LIN {X 0,Y 387.487,Z 857.847,A -85,B 0,C 180,E1 10707.766,E2 10707.766} C_VEL
LIN {X 0,Y 387.621,Z 857.87,A -85,B 0,C 180,E1 10712.229,E2 10712.229} C_VEL
LIN {X 0,Y 387.482,Z 853.741,A -85,B 0,C 180,E1 10716.707,E2 10716.707} C_VEL
LIN {X 0,Y 387.632,Z 843.932,A -85,B 0,C 180,E1 10721.771,E2 10721.771} C_VEL
LIN {X 0,Y 388.622,Z 828.082,A -85,B 0,C 180,E1 10726.928,E2 10726.928} C_VEL
LIN {X 0,Y 390.979,Z 806.956,A -85,B 0,C 180,E1 10731.776,E2 10731.776} C_VEL
LIN {X 0,Y 394.767,Z 780.131,A -85,B 0,C 180,E1 10736.283,E2 10736.283} C_VEL
LIN {X 0,Y 399.363,Z 749.623,A -85,B 0,C 180,E1 10740.039,E2 10740.039} C_VEL
LIN {X 0,Y 404.501,Z 714.96,A -85,B 0,C 180,E1 10743.113,E2 10743.113} C_VEL
LIN {X 0,Y 409.027,Z 678.744,A -85,B 0,C 180,E1 10745.277,E2 10745.277} C_VEL
LIN {X 0,Y 411.733,Z 641.8,A -85,B 0,C 180,E1 10746.674,E2 10746.674} C_VEL
LIN {X 0,Y 397.961,Z 607.635,A -85,B 0,C 180,E1 10748.876,E2 10748.876} C_VEL
LIN {X 0,Y 385.205,Z 581.988,A -85,B 0,C 180,E1 10750.882,E2 10750.882} C_VEL
LIN {X 0,Y 385.096,Z 580.66,A -85,B 0,C 180,E1 10750.941,E2 10750.941} C_VEL
LIN {X 0,Y 385.068,Z 580.66,A -85,B 0,C 180,E1 10758.225,E2 10758.225} C_VEL
LIN {X 0,Y 385.156,Z 580.66,A -85,B 0,C 180,E1 10764.006,E2 10764.006} C_VEL
LIN {X 0,Y 385.319,Z 580.66,A -85,B 0,C 180,E1 10771.967,E2 10771.967} C_VEL
LIN {X 0,Y 385.586,Z 580.66,A -85,B 0,C 180,E1 10779.375,E2 10779.375} C_VEL
LIN {X 0,Y 385.8,Z 580.66,A -85,B 0,C 180,E1 10786.424,E2 10786.424} C_VEL
LIN {X 0,Y 386.219,Z 580.66,A -85,B 0,C 180,E1 10793.265,E2 10793.265} C_VEL
LIN {X 0,Y 386.491,Z 580.66,A -85,B 0,C 180,E1 10799.996,E2 10799.996} C_VEL
LIN {X 0,Y 386.22,Z 580.66,A -85,B 0,C 180,E1 10806.726,E2 10806.726} C_VEL
LIN {X 0,Y 385.936,Z 580.66,A -85,B 0,C 180,E1 10813.562,E2 10813.562} C_VEL
LIN {X 0,Y 385.606,Z 580.66,A -85,B 0,C 180,E1 10820.615,E2 10820.615} C_VEL
LIN {X 0,Y 385.322,Z 580.66,A -85,B 0,C 180,E1 10828.023,E2 10828.023} C_VEL
LIN {X 0,Y 385.109,Z 580.66,A -85,B 0,C 180,E1 10835.989,E2 10835.989} C_VEL
LIN {X 0,Y 385.017,Z 580.66,A -85,B 0,C 180,E1 10841.876,E2 10841.876} C_VEL
LIN {X 0,Y 385.076,Z 580.66,A -85,B 0,C 180,E1 10848.233,E2 10848.233} C_VEL
LIN {X 0,Y 385.211,Z 580.66,A -85,B 0,C 180,E1 10855.382,E2 10855.382} C_VEL
LIN {X 0,Y 398.177,Z 612.723,A -85,B 0,C 180,E1 10858.695,E2 10858.695} C_VEL
LIN {X 0,Y 406.244,Z 641.573,A -85,B 0,C 180,E1 10862.092,E2 10862.092} C_VEL
LIN {X 0,Y 406.168,Z 649.478,A -85,B 0,C 180,E1 10862.96,E2 10862.96} C_VEL
LIN {X 0,Y 401.431,Z 676.101,A -85,B 0,C 180,E1 10866.169,E2 10866.169} C_VEL
LIN {X 0,Y 396.838,Z 698.417,A -85,B 0,C 180,E1 10869.99,E2 10869.99} C_VEL
LIN {X 0,Y 392.904,Z 716.536,A -85,B 0,C 180,E1 10874.407,E2 10874.407} C_VEL
LIN {X 0,Y 390.375,Z 728.782,A -85,B 0,C 180,E1 10878.859,E2 10878.859} C_VEL
LIN {X 0,Y 389.058,Z 736.422,A -85,B 0,C 180,E1 10883.32,E2 10883.32} C_VEL
LIN {X 0,Y 388.574,Z 740.057,A -85,B 0,C 180,E1 10887.776,E2 10887.776} C_VEL
LIN {X 0,Y 388.582,Z 740.014,A -85,B 0,C 180,E1 10892.227,E2 10892.227} C_VEL
LIN {X 0,Y 389.15,Z 736.281,A -85,B 0,C 180,E1 10896.682,E2 10896.682} C_VEL
LIN {X 0,Y 390.68,Z 727.322,A -85,B 0,C 180,E1 10901.701,E2 10901.701} C_VEL
LIN {X 0,Y 393.773,Z 712.297,A -85,B 0,C 180,E1 10906.689,E2 10906.689} C_VEL
LIN {X 0,Y 398.048,Z 692.52,A -85,B 0,C 180,E1 10911.054,E2 10911.054} C_VEL
LIN {X 0,Y 402.806,Z 668.479,A -85,B 0,C 180,E1 10914.779,E2 10914.779} C_VEL
LIN {X 0,Y 406.697,Z 643.345,A -85,B 0,C 180,E1 10917.577,E2 10917.577} C_VEL
LIN {X 0,Y 398.963,Z 615.178,A -85,B 0,C 180,E1 10920.925,E2 10920.925} C_VEL
LIN {X 0,Y 386.913,Z 585.522,A -85,B 0,C 180,E1 10924.088,E2 10924.088} C_VEL
LIN {X 0,Y 385.16,Z 580.66,A -85,B 0,C 180,E1 10924.654,E2 10924.654} C_VEL
LIN {X 0,Y 385.049,Z 580.66,A -85,B 0,C 180,E1 10931.776,E2 10931.776} C_VEL
LIN {X 0,Y 385.058,Z 580.66,A -85,B 0,C 180,E1 10938.235,E2 10938.235} C_VEL
LIN {X 0,Y 385.139,Z 580.66,A -85,B 0,C 180,E1 10944.014,E2 10944.014} C_VEL
LIN {X 0,Y 385.264,Z 580.66,A -85,B 0,C 180,E1 10951.972,E2 10951.972} C_VEL
LIN {X 0,Y 385.581,Z 580.66,A -85,B 0,C 180,E1 10959.383,E2 10959.383} C_VEL
LIN {X 0,Y 385.746,Z 580.66,A -85,B 0,C 180,E1 10966.431,E2 10966.431} C_VEL
LIN {X 0,Y 386.233,Z 580.66,A -85,B 0,C 180,E1 10973.274,E2 10973.274} C_VEL
LIN {X 0,Y 386.501,Z 580.66,A -85,B 0,C 180,E1 10980.004,E2 10980.004} C_VEL
LIN {X 0,Y 386.216,Z 580.66,A -85,B 0,C 180,E1 10986.735,E2 10986.735} C_VEL
LIN {X 0,Y 385.929,Z 580.66,A -85,B 0,C 180,E1 10993.571,E2 10993.571} C_VEL
LIN {X 0,Y 385.585,Z 580.66,A -85,B 0,C 180,E1 11000.626,E2 11000.626} C_VEL
LIN {X 0,Y 385.302,Z 580.66,A -85,B 0,C 180,E1 11008.034,E2 11008.034} C_VEL
LIN {X 0,Y 385.067,Z 580.66,A -85,B 0,C 180,E1 11014.62,E2 11014.62} C_VEL
LIN {X 0,Y 385.011,Z 580.66,A -85,B 0,C 180,E1 11021.782,E2 11021.782} C_VEL
LIN {X 0,Y 385.175,Z 580.66,A -85,B 0,C 180,E1 11029.063,E2 11029.063} C_VEL
LIN {X 0,Y 407.62,Z 629.809,A -85,B 0,C 180,E1 11032.612,E2 11032.612} C_VEL
LIN {X 0,Y 412.212,Z 644.181,A -85,B 0,C 180,E1 11033.455,E2 11033.455} C_VEL
LIN {X 0,Y 408.523,Z 682.741,A -85,B 0,C 180,E1 11034.911,E2 11034.911} C_VEL
LIN {X 0,Y 403.964,Z 718.267,A -85,B 0,C 180,E1 11037.144,E2 11037.144} C_VEL
LIN {X 0,Y 398.982,Z 752.199,A -85,B 0,C 180,E1 11040.237,E2 11040.237} C_VEL
LIN {X 0,Y 394.303,Z 783.048,A -85,B 0,C 180,E1 11044.15,E2 11044.15} C_VEL
LIN {X 0,Y 390.715,Z 809.2,A -85,B 0,C 180,E1 11048.674,E2 11048.674} C_VEL
LIN {X 0,Y 388.558,Z 830.209,A -85,B 0,C 180,E1 11053.646,E2 11053.646} C_VEL
LIN {X 0,Y 387.619,Z 845.23,A -85,B 0,C 180,E1 11058.774,E2 11058.774} C_VEL
LIN {X 0,Y 387.505,Z 852.985,A -85,B 0,C 180,E1 11062.805,E2 11062.805} C_VEL
LIN {X 0,Y 385.019,Z 855.196,A -85,B 0,C 180,E1 11064.686,E2 11064.686} C_VEL
LIN {X 0,Y 379.649,Z 856.7,A -85,B 0,C 180,E1 11067.891,E2 11067.891} C_VEL
LIN {X 0,Y 379.794,Z 856.679,A -85,B 0,C 180,E1 11072.275,E2 11072.275} C_VEL
LIN {X 0,Y 379.657,Z 852.534,A -85,B 0,C 180,E1 11076.846,E2 11076.846} C_VEL
LIN {X 0,Y 379.775,Z 842.813,A -85,B 0,C 180,E1 11081.967,E2 11081.967} C_VEL
LIN {X 0,Y 380.838,Z 827.231,A -85,B 0,C 180,E1 11087.164,E2 11087.164} C_VEL
LIN {X 0,Y 383.309,Z 806.131,A -85,B 0,C 180,E1 11092.126,E2 11092.126} C_VEL
LIN {X 0,Y 387.248,Z 779.805,A -85,B 0,C 180,E1 11096.668,E2 11096.668} C_VEL
LIN {X 0,Y 392.071,Z 749.47,A -85,B 0,C 180,E1 11100.497,E2 11100.497} C_VEL
LIN {X 0,Y 397.304,Z 715.923,A -85,B 0,C 180,E1 11103.556,E2 11103.556} C_VEL
LIN {X 0,Y 402.117,Z 679.727,A -85,B 0,C 180,E1 11105.805,E2 11105.805} C_VEL
LIN {X 0,Y 405.031,Z 644.006,A -85,B 0,C 180,E1 11107.216,E2 11107.216} C_VEL
LIN {X 0,Y 392.035,Z 611.501,A -85,B 0,C 180,E1 11109.406,E2 11109.406} C_VEL
LIN {X 0,Y 377.128,Z 580.66,A -85,B 0,C 180,E1 11111.91,E2 11111.91} C_VEL
LIN {X 0,Y 377.101,Z 580.66,A -85,B 0,C 180,E1 11119.484,E2 11119.484} C_VEL
LIN {X 0,Y 377.196,Z 580.66,A -85,B 0,C 180,E1 11125.937,E2 11125.937} C_VEL
LIN {X 0,Y 377.413,Z 580.66,A -85,B 0,C 180,E1 11133.906,E2 11133.906} C_VEL
LIN {X 0,Y 377.618,Z 580.66,A -85,B 0,C 180,E1 11138.919,E2 11138.919} C_VEL
LIN {X 0,Y 377.856,Z 580.66,A -85,B 0,C 180,E1 11146.133,E2 11146.133} C_VEL
LIN {X 0,Y 378.293,Z 580.66,A -85,B 0,C 180,E1 11153.123,E2 11153.123} C_VEL
LIN {X 0,Y 378.59,Z 580.66,A -85,B 0,C 180,E1 11159.996,E2 11159.996} C_VEL
LIN {X 0,Y 378.296,Z 580.66,A -85,B 0,C 180,E1 11166.868,E2 11166.868} C_VEL
LIN {X 0,Y 377.984,Z 580.66,A -85,B 0,C 180,E1 11173.853,E2 11173.853} C_VEL
LIN {X 0,Y 377.637,Z 580.66,A -85,B 0,C 180,E1 11181.071,E2 11181.071} C_VEL
LIN {X 0,Y 377.334,Z 580.66,A -85,B 0,C 180,E1 11188.671,E2 11188.671} C_VEL
LIN {X 0,Y 377.167,Z 580.66,A -85,B 0,C 180,E1 11194.056,E2 11194.056} C_VEL
LIN {X 0,Y 377.046,Z 580.66,A -85,B 0,C 180,E1 11200.506,E2 11200.506} C_VEL
LIN {X 0,Y 377.061,Z 580.66,A -85,B 0,C 180,E1 11207.135,E2 11207.135} C_VEL
LIN {X 0,Y 377.268,Z 581.284,A -85,B 0,C 180,E1 11214.461,E2 11214.461} C_VEL
LIN {X 0,Y 390.662,Z 613.094,A -85,B 0,C 180,E1 11217.911,E2 11217.911} C_VEL
LIN {X 0,Y 398.837,Z 642.106,A -85,B 0,C 180,E1 11221.418,E2 11221.418} C_VEL
LIN {X 0,Y 399.58,Z 649.041,A -85,B 0,C 180,E1 11222.269,E2 11222.269} C_VEL
LIN {X 0,Y 394.701,Z 675.471,A -85,B 0,C 180,E1 11225.436,E2 11225.436} C_VEL
LIN {X 0,Y 389.766,Z 698.393,A -85,B 0,C 180,E1 11229.334,E2 11229.334} C_VEL
LIN {X 0,Y 385.74,Z 716.002,A -85,B 0,C 180,E1 11233.577,E2 11233.577} C_VEL
LIN {X 0,Y 382.702,Z 729.982,A -85,B 0,C 180,E1 11238.632,E2 11238.632} C_VEL
LIN {X 0,Y 381.313,Z 737.611,A -85,B 0,C 180,E1 11243.184,E2 11243.184} C_VEL
LIN {X 0,Y 380.788,Z 741.241,A -85,B 0,C 180,E1 11247.731,E2 11247.731} C_VEL
LIN {X 0,Y 380.797,Z 741.198,A -85,B 0,C 180,E1 11252.273,E2 11252.273} C_VEL
LIN {X 0,Y 381.602,Z 736.01,A -85,B 0,C 180,E1 11257.918,E2 11257.918} C_VEL
LIN {X 0,Y 383.654,Z 725.73,A -85,B 0,C 180,E1 11263.072,E2 11263.072} C_VEL
LIN {X 0,Y 387.075,Z 710.25,A -85,B 0,C 180,E1 11267.876,E2 11267.876} C_VEL
LIN {X 0,Y 391.675,Z 689.835,A -85,B 0,C 180,E1 11272.192,E2 11272.192} C_VEL
LIN {X 0,Y 396.785,Z 664.357,A -85,B 0,C 180,E1 11275.936,E2 11275.936} C_VEL
LIN {X 0,Y 399.548,Z 645.168,A -85,B 0,C 180,E1 11278.079,E2 11278.079} C_VEL
LIN {X 0,Y 391.906,Z 617.092,A -85,B 0,C 180,E1 11281.529,E2 11281.529} C_VEL
LIN {X 0,Y 380.331,Z 588.674,A -85,B 0,C 180,E1 11284.708,E2 11284.708} C_VEL
LIN {X 0,Y 377.226,Z 580.66,A -85,B 0,C 180,E1 11285.614,E2 11285.614} C_VEL
LIN {X 0,Y 377.045,Z 580.66,A -85,B 0,C 180,E1 11292.872,E2 11292.872} C_VEL
LIN {X 0,Y 377.104,Z 580.66,A -85,B 0,C 180,E1 11300.2,E2 11300.2} C_VEL
LIN {X 0,Y 377.171,Z 580.66,A -85,B 0,C 180,E1 11307.157,E2 11307.157} C_VEL
LIN {X 0,Y 377.374,Z 580.66,A -85,B 0,C 180,E1 11313.913,E2 11313.913} C_VEL
LIN {X 0,Y 377.61,Z 580.66,A -85,B 0,C 180,E1 11318.928,E2 11318.928} C_VEL
LIN {X 0,Y 377.805,Z 580.66,A -85,B 0,C 180,E1 11326.14,E2 11326.14} C_VEL
LIN {X 0,Y 378.304,Z 580.66,A -85,B 0,C 180,E1 11333.155,E2 11333.155} C_VEL
LIN {X 0,Y 378.599,Z 580.66,A -85,B 0,C 180,E1 11340.004,E2 11340.004} C_VEL
LIN {X 0,Y 378.299,Z 580.66,A -85,B 0,C 180,E1 11346.877,E2 11346.877} C_VEL
LIN {X 0,Y 377.979,Z 580.66,A -85,B 0,C 180,E1 11353.862,E2 11353.862} C_VEL
LIN {X 0,Y 377.616,Z 580.66,A -85,B 0,C 180,E1 11361.081,E2 11361.081} C_VEL
LIN {X 0,Y 377.338,Z 580.66,A -85,B 0,C 180,E1 11368.68,E2 11368.68} C_VEL
LIN {X 0,Y 377.161,Z 580.66,A -85,B 0,C 180,E1 11374.067,E2 11374.067} C_VEL
LIN {X 0,Y 377.026,Z 580.66,A -85,B 0,C 180,E1 11380.497,E2 11380.497} C_VEL
LIN {X 0,Y 377.195,Z 580.872,A -85,B 0,C 180,E1 11388.16,E2 11388.16} C_VEL
LIN {X 0,Y 386.408,Z 599.748,A -85,B 0,C 180,E1 11389.706,E2 11389.706} C_VEL
LIN {X 0,Y 403.016,Z 637.674,A -85,B 0,C 180,E1 11392.386,E2 11392.386} C_VEL
LIN {X 0,Y 405.397,Z 647.401,A -85,B 0,C 180,E1 11392.942,E2 11392.942} C_VEL
LIN {X 0,Y 401.341,Z 685.437,A -85,B 0,C 180,E1 11394.49,E2 11394.49} C_VEL
LIN {X 0,Y 396.408,Z 721.378,A -85,B 0,C 180,E1 11396.873,E2 11396.873} C_VEL
LIN {X 0,Y 391.163,Z 755.108,A -85,B 0,C 180,E1 11400.13,E2 11400.13} C_VEL
LIN {X 0,Y 386.341,Z 785.338,A -85,B 0,C 180,E1 11404.188,E2 11404.188} C_VEL
LIN {X 0,Y 382.632,Z 811.449,A -85,B 0,C 180,E1 11408.978,E2 11408.978} C_VEL
LIN {X 0,Y 380.581,Z 830.851,A -85,B 0,C 180,E1 11413.885,E2 11413.885} C_VEL
LIN {X 0,Y 379.721,Z 845.274,A -85,B 0,C 180,E1 11419.118,E2 11419.118} C_VEL
LIN {X 0,Y 379.676,Z 852.977,A -85,B 0,C 180,E1 11423.511,E2 11423.511} C_VEL
LIN {X 0,Y 379.649,Z 856.7,A -85,B 0,C 180,E1 11427.891,E2 11427.891} C_VEL
LIN {X 0,Y 377.151,Z 856.83,A -85,B 0,C 180,E1 11429.837,E2 11429.837} C_VEL
LIN {X 0,Y 371.879,Z 854.962,A -85,B 0,C 180,E1 11433.101,E2 11433.101} C_VEL
LIN {X 0,Y 371.822,Z 849.562,A -85,B 0,C 180,E1 11438.164,E2 11438.164} C_VEL
LIN {X 0,Y 372.107,Z 838.206,A -85,B 0,C 180,E1 11443.558,E2 11443.558} C_VEL
LIN {X 0,Y 373.57,Z 821.118,A -85,B 0,C 180,E1 11448.85,E2 11448.85} C_VEL
LIN {X 0,Y 376.666,Z 798.023,A -85,B 0,C 180,E1 11453.927,E2 11453.927} C_VEL
LIN {X 0,Y 381.131,Z 770.539,A -85,B 0,C 180,E1 11458.363,E2 11458.363} C_VEL
LIN {X 0,Y 386.638,Z 738.34,A -85,B 0,C 180,E1 11462.121,E2 11462.121} C_VEL
LIN {X 0,Y 392.059,Z 704.385,A -85,B 0,C 180,E1 11464.934,E2 11464.934} C_VEL
LIN {X 0,Y 396.892,Z 667.975,A -85,B 0,C 180,E1 11466.93,E2 11466.93} C_VEL
LIN {X 0,Y 398.263,Z 645.749,A -85,B 0,C 180,E1 11467.803,E2 11467.803} C_VEL
LIN {X 0,Y 385.396,Z 613.636,A -85,B 0,C 180,E1 11470.079,E2 11470.079} C_VEL
LIN {X 0,Y 369.227,Z 581.844,A -85,B 0,C 180,E1 11472.825,E2 11472.825} C_VEL
LIN {X 0,Y 369.134,Z 580.66,A -85,B 0,C 180,E1 11472.996,E2 11472.996} C_VEL
LIN {X 0,Y 369.156,Z 580.66,A -85,B 0,C 180,E1 11479.152,E2 11479.152} C_VEL
LIN {X 0,Y 369.201,Z 580.66,A -85,B 0,C 180,E1 11485.094,E2 11485.094} C_VEL
LIN {X 0,Y 369.331,Z 580.66,A -85,B 0,C 180,E1 11490.638,E2 11490.638} C_VEL
LIN {X 0,Y 369.537,Z 580.66,A -85,B 0,C 180,E1 11495.896,E2 11495.896} C_VEL
LIN {X 0,Y 369.846,Z 580.66,A -85,B 0,C 180,E1 11503.402,E2 11503.402} C_VEL
LIN {X 0,Y 370.128,Z 580.66,A -85,B 0,C 180,E1 11510.611,E2 11510.611} C_VEL
LIN {X 0,Y 370.709,Z 580.66,A -85,B 0,C 180,E1 11517.663,E2 11517.663} C_VEL
LIN {X 0,Y 370.608,Z 580.66,A -85,B 0,C 180,E1 11524.666,E2 11524.666} C_VEL
LIN {X 0,Y 370.124,Z 580.66,A -85,B 0,C 180,E1 11531.932,E2 11531.932} C_VEL
LIN {X 0,Y 369.775,Z 580.66,A -85,B 0,C 180,E1 11539.048,E2 11539.048} C_VEL
LIN {X 0,Y 369.457,Z 580.66,A -85,B 0,C 180,E1 11546.69,E2 11546.69} C_VEL
LIN {X 0,Y 369.278,Z 580.66,A -85,B 0,C 180,E1 11552.08,E2 11552.08} C_VEL
LIN {X 0,Y 369.09,Z 580.66,A -85,B 0,C 180,E1 11559.038,E2 11559.038} C_VEL
LIN {X 0,Y 369.142,Z 580.66,A -85,B 0,C 180,E1 11565.984,E2 11565.984} C_VEL
LIN {X 0,Y 369.295,Z 580.686,A -85,B 0,C 180,E1 11573.414,E2 11573.414} C_VEL
LIN {X 0,Y 382.702,Z 612.445,A -85,B 0,C 180,E1 11576.965,E2 11576.965} C_VEL
LIN {X 0,Y 390.981,Z 640.632,A -85,B 0,C 180,E1 11580.443,E2 11580.443} C_VEL
LIN {X 0,Y 392.512,Z 651.519,A -85,B 0,C 180,E1 11581.853,E2 11581.853} C_VEL
LIN {X 0,Y 387.224,Z 678.672,A -85,B 0,C 180,E1 11585.237,E2 11585.237} C_VEL
LIN {X 0,Y 382.184,Z 700.911,A -85,B 0,C 180,E1 11589.188,E2 11589.188} C_VEL
LIN {X 0,Y 377.843,Z 718.965,A -85,B 0,C 180,E1 11593.769,E2 11593.769} C_VEL
LIN {X 0,Y 374.79,Z 732.393,A -85,B 0,C 180,E1 11598.977,E2 11598.977} C_VEL
LIN {X 0,Y 373.319,Z 740.078,A -85,B 0,C 180,E1 11604.202,E2 11604.202} C_VEL
LIN {X 0,Y 372.998,Z 742.425,A -85,B 0,C 180,E1 11607.683,E2 11607.683} C_VEL
LIN {X 0,Y 373.007,Z 742.383,A -85,B 0,C 180,E1 11612.32,E2 11612.32} C_VEL
LIN {X 0,Y 373.813,Z 737.617,A -85,B 0,C 180,E1 11617.804,E2 11617.804} C_VEL
LIN {X 0,Y 376.06,Z 726.932,A -85,B 0,C 180,E1 11623.341,E2 11623.341} C_VEL
LIN {X 0,Y 379.463,Z 712.313,A -85,B 0,C 180,E1 11628.022,E2 11628.022} C_VEL
LIN {X 0,Y 384.164,Z 692.319,A -85,B 0,C 180,E1 11632.405,E2 11632.405} C_VEL
LIN {X 0,Y 389.405,Z 667.874,A -85,B 0,C 180,E1 11636.155,E2 11636.155} C_VEL
LIN {X 0,Y 392.524,Z 647.521,A -85,B 0,C 180,E1 11638.527,E2 11638.527} C_VEL
LIN {X 0,Y 384.969,Z 619.184,A -85,B 0,C 180,E1 11642.131,E2 11642.131} C_VEL
LIN {X 0,Y 373.521,Z 590.683,A -85,B 0,C 180,E1 11645.441,E2 11645.441} C_VEL
LIN {X 0,Y 369.288,Z 580.66,A -85,B 0,C 180,E1 11646.597,E2 11646.597} C_VEL
LIN {X 0,Y 369.139,Z 580.66,A -85,B 0,C 180,E1 11654.022,E2 11654.022} C_VEL
LIN {X 0,Y 369.13,Z 580.66,A -85,B 0,C 180,E1 11660.96,E2 11660.96} C_VEL
LIN {X 0,Y 369.253,Z 580.66,A -85,B 0,C 180,E1 11667.918,E2 11667.918} C_VEL
LIN {X 0,Y 369.513,Z 580.66,A -85,B 0,C 180,E1 11675.904,E2 11675.904} C_VEL
LIN {X 0,Y 369.746,Z 580.66,A -85,B 0,C 180,E1 11680.95,E2 11680.95} C_VEL
LIN {X 0,Y 369.994,Z 580.66,A -85,B 0,C 180,E1 11688.239,E2 11688.239} C_VEL
LIN {X 0,Y 370.488,Z 580.66,A -85,B 0,C 180,E1 11695.332,E2 11695.332} C_VEL
LIN {X 0,Y 370.722,Z 580.66,A -85,B 0,C 180,E1 11700.004,E2 11700.004} C_VEL
LIN {X 0,Y 370.369,Z 580.66,A -85,B 0,C 180,E1 11707.025,E2 11707.025} C_VEL
LIN {X 0,Y 370.037,Z 580.66,A -85,B 0,C 180,E1 11714.166,E2 11714.166} C_VEL
LIN {X 0,Y 369.677,Z 580.66,A -85,B 0,C 180,E1 11721.556,E2 11721.556} C_VEL
LIN {X 0,Y 369.456,Z 580.66,A -85,B 0,C 180,E1 11726.7,E2 11726.7} C_VEL
LIN {X 0,Y 369.268,Z 580.66,A -85,B 0,C 180,E1 11732.091,E2 11732.091} C_VEL
LIN {X 0,Y 369.058,Z 580.66,A -85,B 0,C 180,E1 11739.026,E2 11739.026} C_VEL
LIN {X 0,Y 369.152,Z 580.66,A -85,B 0,C 180,E1 11745.98,E2 11745.98} C_VEL
LIN {X 0,Y 369.209,Z 581.4,A -85,B 0,C 180,E1 11747.179,E2 11747.179} C_VEL
LIN {X 0,Y 391.31,Z 626.732,A -85,B 0,C 180,E1 11750.903,E2 11750.903} C_VEL
LIN {X 0,Y 398.754,Z 648.256,A -85,B 0,C 180,E1 11752.346,E2 11752.346} C_VEL
LIN {X 0,Y 394.452,Z 686.258,A -85,B 0,C 180,E1 11753.954,E2 11753.954} C_VEL
LIN {X 0,Y 389.256,Z 722.076,A -85,B 0,C 180,E1 11756.401,E2 11756.401} C_VEL
LIN {X 0,Y 383.757,Z 755.406,A -85,B 0,C 180,E1 11759.728,E2 11759.728} C_VEL
LIN {X 0,Y 378.743,Z 785.057,A -85,B 0,C 180,E1 11763.818,E2 11763.818} C_VEL
LIN {X 0,Y 374.823,Z 811.132,A -85,B 0,C 180,E1 11768.756,E2 11768.756} C_VEL
LIN {X 0,Y 372.615,Z 831.492,A -85,B 0,C 180,E1 11774.135,E2 11774.135} C_VEL
LIN {X 0,Y 371.851,Z 845.324,A -85,B 0,C 180,E1 11779.477,E2 11779.477} C_VEL
LIN {X 0,Y 371.849,Z 852.304,A -85,B 0,C 180,E1 11783.824,E2 11783.824} C_VEL
LIN {X 0,Y 371.828,Z 855.519,A -85,B 0,C 180,E1 11787.884,E2 11787.884} C_VEL
LIN {X 0,Y 371.967,Z 855.488,A -85,B 0,C 180,E1 11792.323,E2 11792.323} C_VEL
LIN {X 0,Y 371.879,Z 854.962,A -85,B 0,C 180,E1 11793.101,E2 11793.101} C_VEL
LIN {X 0,Y 369.293,Z 853.192,A -85,B 0,C 180,E1 11795.068,E2 11795.068} C_VEL
LIN {X 0,Y 364.056,Z 848.87,A -85,B 0,C 180,E1 11797.999,E2 11797.999} C_VEL
LIN {X 0,Y 363.982,Z 848.354,A -85,B 0,C 180,E1 11798.338,E2 11798.338} C_VEL
LIN {X 0,Y 364.281,Z 836.657,A -85,B 0,C 180,E1 11803.975,E2 11803.975} C_VEL
LIN {X 0,Y 366.051,Z 818.641,A -85,B 0,C 180,E1 11809.566,E2 11809.566} C_VEL
LIN {X 0,Y 369.486,Z 795.121,A -85,B 0,C 180,E1 11814.744,E2 11814.744} C_VEL
LIN {X 0,Y 374.437,Z 766.272,A -85,B 0,C 180,E1 11819.346,E2 11819.346} C_VEL
LIN {X 0,Y 380.177,Z 733.933,A -85,B 0,C 180,E1 11823.073,E2 11823.073} C_VEL
LIN {X 0,Y 386.003,Z 698.709,A -85,B 0,C 180,E1 11825.897,E2 11825.897} C_VEL
LIN {X 0,Y 390.728,Z 663.112,A -85,B 0,C 180,E1 11827.761,E2 11827.761} C_VEL
LIN {X 0,Y 391.645,Z 647.863,A -85,B 0,C 180,E1 11828.377,E2 11828.377} C_VEL
LIN {X 0,Y 378.919,Z 616.13,A -85,B 0,C 180,E1 11830.754,E2 11830.754} C_VEL
LIN {X 0,Y 361.299,Z 581.694,A -85,B 0,C 180,E1 11833.878,E2 11833.878} C_VEL
LIN {X 0,Y 361.227,Z 580.66,A -85,B 0,C 180,E1 11833.994,E2 11833.994} C_VEL
LIN {X 0,Y 361.234,Z 580.66,A -85,B 0,C 180,E1 11841.199,E2 11841.199} C_VEL
LIN {X 0,Y 361.277,Z 580.66,A -85,B 0,C 180,E1 11847.111,E2 11847.111} C_VEL
LIN {X 0,Y 361.455,Z 580.66,A -85,B 0,C 180,E1 11852.66,E2 11852.66} C_VEL
LIN {X 0,Y 361.69,Z 580.66,A -85,B 0,C 180,E1 11857.943,E2 11857.943} C_VEL
LIN {X 0,Y 361.979,Z 580.66,A -85,B 0,C 180,E1 11865.512,E2 11865.512} C_VEL
LIN {X 0,Y 362.435,Z 580.66,A -85,B 0,C 180,E1 11872.821,E2 11872.821} C_VEL
LIN {X 0,Y 362.812,Z 580.66,A -85,B 0,C 180,E1 11879.996,E2 11879.996} C_VEL
LIN {X 0,Y 362.445,Z 580.66,A -85,B 0,C 180,E1 11887.17,E2 11887.17} C_VEL
LIN {X 0,Y 362.1,Z 580.66,A -85,B 0,C 180,E1 11894.474,E2 11894.474} C_VEL
LIN {X 0,Y 361.707,Z 580.66,A -85,B 0,C 180,E1 11902.046,E2 11902.046} C_VEL
LIN {X 0,Y 361.385,Z 580.66,A -85,B 0,C 180,E1 11908.742,E2 11908.742} C_VEL
LIN {X 0,Y 361.178,Z 580.66,A -85,B 0,C 180,E1 11915.788,E2 11915.788} C_VEL
LIN {X 0,Y 361.179,Z 580.66,A -85,B 0,C 180,E1 11921.939,E2 11921.939} C_VEL
LIN {X 0,Y 361.251,Z 580.66,A -85,B 0,C 180,E1 11928.741,E2 11928.741} C_VEL
LIN {X 0,Y 361.288,Z 580.699,A -85,B 0,C 180,E1 11932.329,E2 11932.329} C_VEL
LIN {X 0,Y 375.138,Z 612.697,A -85,B 0,C 180,E1 11936.083,E2 11936.083} C_VEL
LIN {X 0,Y 383.173,Z 639.476,A -85,B 0,C 180,E1 11939.471,E2 11939.471} C_VEL
LIN {X 0,Y 385.708,Z 652.742,A -85,B 0,C 180,E1 11941.292,E2 11941.292} C_VEL
LIN {X 0,Y 380.178,Z 679.949,A -85,B 0,C 180,E1 11944.746,E2 11944.746} C_VEL
LIN {X 0,Y 374.903,Z 702.152,A -85,B 0,C 180,E1 11948.765,E2 11948.765} C_VEL
LIN {X 0,Y 370.327,Z 720.178,A -85,B 0,C 180,E1 11953.43,E2 11953.43} C_VEL
LIN {X 0,Y 367.119,Z 733.591,A -85,B 0,C 180,E1 11958.744,E2 11958.744} C_VEL
LIN {X 0,Y 365.55,Z 741.266,A -85,B 0,C 180,E1 11964.079,E2 11964.079} C_VEL
LIN {X 0,Y 365.212,Z 743.609,A -85,B 0,C 180,E1 11967.634,E2 11967.634} C_VEL
LIN {X 0,Y 365.222,Z 743.567,A -85,B 0,C 180,E1 11972.37,E2 11972.37} C_VEL
LIN {X 0,Y 365.884,Z 739.855,A -85,B 0,C 180,E1 11977.109,E2 11977.109} C_VEL
LIN {X 0,Y 367.748,Z 730.936,A -85,B 0,C 180,E1 11982.442,E2 11982.442} C_VEL
LIN {X 0,Y 371.34,Z 716.166,A -85,B 0,C 180,E1 11987.666,E2 11987.666} C_VEL
LIN {X 0,Y 376.133,Z 697.11,A -85,B 0,C 180,E1 11992.177,E2 11992.177} C_VEL
LIN {X 0,Y 381.475,Z 673.599,A -85,B 0,C 180,E1 11996.079,E2 11996.079} C_VEL
LIN {X 0,Y 385.666,Z 650.724,A -85,B 0,C 180,E1 11998.858,E2 11998.858} C_VEL
LIN {X 0,Y 378.791,Z 623.486,A -85,B 0,C 180,E1 12002.486,E2 12002.486} C_VEL
LIN {X 0,Y 367.612,Z 594.962,A -85,B 0,C 180,E1 12005.96,E2 12005.96} C_VEL
LIN {X 0,Y 361.269,Z 580.66,A -85,B 0,C 180,E1 12007.578,E2 12007.578} C_VEL
LIN {X 0,Y 361.217,Z 580.66,A -85,B 0,C 180,E1 12015.249,E2 12015.249} C_VEL
LIN {X 0,Y 361.206,Z 580.66,A -85,B 0,C 180,E1 12022.537,E2 12022.537} C_VEL
LIN {X 0,Y 361.358,Z 580.66,A -85,B 0,C 180,E1 12029.935,E2 12029.935} C_VEL
LIN {X 0,Y 361.679,Z 580.66,A -85,B 0,C 180,E1 12037.952,E2 12037.952} C_VEL
LIN {X 0,Y 361.918,Z 580.66,A -85,B 0,C 180,E1 12045.519,E2 12045.519} C_VEL
LIN {X 0,Y 362.43,Z 580.66,A -85,B 0,C 180,E1 12053.135,E2 12053.135} C_VEL
LIN {X 0,Y 362.819,Z 580.66,A -85,B 0,C 180,E1 12060.004,E2 12060.004} C_VEL
LIN {X 0,Y 362.455,Z 580.66,A -85,B 0,C 180,E1 12067.179,E2 12067.179} C_VEL
LIN {X 0,Y 362.082,Z 580.66,A -85,B 0,C 180,E1 12074.484,E2 12074.484} C_VEL
LIN {X 0,Y 361.69,Z 580.66,A -85,B 0,C 180,E1 12082.057,E2 12082.057} C_VEL
LIN {X 0,Y 361.385,Z 580.66,A -85,B 0,C 180,E1 12090.073,E2 12090.073} C_VEL
LIN {X 0,Y 361.146,Z 580.66,A -85,B 0,C 180,E1 12097.45,E2 12097.45} C_VEL
LIN {X 0,Y 361.193,Z 580.66,A -85,B 0,C 180,E1 12104.747,E2 12104.747} C_VEL
LIN {X 0,Y 361.282,Z 581.215,A -85,B 0,C 180,E1 12106.126,E2 12106.126} C_VEL
LIN {X 0,Y 383.637,Z 626.463,A -85,B 0,C 180,E1 12110.068,E2 12110.068} C_VEL
LIN {X 0,Y 391.968,Z 649.234,A -85,B 0,C 180,E1 12111.726,E2 12111.726} C_VEL
LIN {X 0,Y 387.707,Z 686.192,A -85,B 0,C 180,E1 12113.347,E2 12113.347} C_VEL
LIN {X 0,Y 382.165,Z 722.435,A -85,B 0,C 180,E1 12115.886,E2 12115.886} C_VEL
LIN {X 0,Y 376.285,Z 756.1,A -85,B 0,C 180,E1 12119.356,E2 12119.356} C_VEL
LIN {X 0,Y 371.185,Z 784.787,A -85,B 0,C 180,E1 12123.436,E2 12123.436} C_VEL
LIN {X 0,Y 367.2,Z 809.818,A -85,B 0,C 180,E1 12128.293,E2 12128.293} C_VEL
LIN {X 0,Y 364.984,Z 828.294,A -85,B 0,C 180,E1 12133.176,E2 12133.176} C_VEL
LIN {X 0,Y 364.039,Z 842.803,A -85,B 0,C 180,E1 12138.643,E2 12138.643} C_VEL
LIN {X 0,Y 364.02,Z 850.112,A -85,B 0,C 180,E1 12142.855,E2 12142.855} C_VEL
LIN {X 0,Y 364.024,Z 854.276,A -85,B 0,C 180,E1 12147.622,E2 12147.622} C_VEL
LIN {X 0,Y 364.14,Z 854.297,A -85,B 0,C 180,E1 12152.373,E2 12152.373} C_VEL
LIN {X 0,Y 363.996,Z 850.12,A -85,B 0,C 180,E1 12157.142,E2 12157.142} C_VEL
LIN {X 0,Y 363.982,Z 848.354,A -85,B 0,C 180,E1 12158.338,E2 12158.338} C_VEL
LIN {X 0,Y 361.535,Z 844.791,A -85,B 0,C 180,E1 12160.295,E2 12160.295} C_VEL
LIN {X 0,Y 356.399,Z 838.109,A -85,B 0,C 180,E1 12163.178,E2 12163.178} C_VEL
LIN {X 0,Y 356.353,Z 837.297,A -85,B 0,C 180,E1 12163.509,E2 12163.509} C_VEL
LIN {X 0,Y 357.9,Z 820.394,A -85,B 0,C 180,E1 12169.186,E2 12169.186} C_VEL
LIN {X 0,Y 361.501,Z 796.939,A -85,B 0,C 180,E1 12174.668,E2 12174.668} C_VEL
LIN {X 0,Y 366.338,Z 769.814,A -85,B 0,C 180,E1 12179.281,E2 12179.281} C_VEL
LIN {X 0,Y 372.334,Z 738.262,A -85,B 0,C 180,E1 12183.166,E2 12183.166} C_VEL
LIN {X 0,Y 378.164,Z 705.17,A -85,B 0,C 180,E1 12186.051,E2 12186.051} C_VEL
LIN {X 0,Y 383.426,Z 669.623,A -85,B 0,C 180,E1 12188.129,E2 12188.129} C_VEL
LIN {X 0,Y 384.867,Z 649.638,A -85,B 0,C 180,E1 12188.992,E2 12188.992} C_VEL
LIN {X 0,Y 371.618,Z 616.677,A -85,B 0,C 180,E1 12191.611,E2 12191.611} C_VEL
LIN {X 0,Y 353.37,Z 581.449,A -85,B 0,C 180,E1 12195,E2 12195} C_VEL
LIN {X 0,Y 353.28,Z 580.66,A -85,B 0,C 180,E1 12200.244,E2 12200.244} C_VEL
LIN {X 0,Y 353.32,Z 580.66,A -85,B 0,C 180,E1 12206.272,E2 12206.272} C_VEL
LIN {X 0,Y 353.522,Z 580.66,A -85,B 0,C 180,E1 12213.675,E2 12213.675} C_VEL
LIN {X 0,Y 353.833,Z 580.66,A -85,B 0,C 180,E1 12220.048,E2 12220.048} C_VEL
LIN {X 0,Y 354.188,Z 580.66,A -85,B 0,C 180,E1 12227.697,E2 12227.697} C_VEL
LIN {X 0,Y 354.647,Z 580.66,A -85,B 0,C 180,E1 12235.114,E2 12235.114} C_VEL
LIN {X 0,Y 354.916,Z 580.66,A -85,B 0,C 180,E1 12239.995,E2 12239.995} C_VEL
LIN {X 0,Y 354.51,Z 580.66,A -85,B 0,C 180,E1 12247.331,E2 12247.331} C_VEL
LIN {X 0,Y 354.165,Z 580.66,A -85,B 0,C 180,E1 12254.806,E2 12254.806} C_VEL
LIN {X 0,Y 353.766,Z 580.66,A -85,B 0,C 180,E1 12262.568,E2 12262.568} C_VEL
LIN {X 0,Y 353.493,Z 580.66,A -85,B 0,C 180,E1 12267.998,E2 12267.998} C_VEL
LIN {X 0,Y 353.292,Z 580.66,A -85,B 0,C 180,E1 12275.761,E2 12275.761} C_VEL
LIN {X 0,Y 353.185,Z 580.66,A -85,B 0,C 180,E1 12283.427,E2 12283.427} C_VEL
LIN {X 0,Y 353.361,Z 580.66,A -85,B 0,C 180,E1 12291.145,E2 12291.145} C_VEL
LIN {X 0,Y 367.608,Z 613.079,A -85,B 0,C 180,E1 12295.168,E2 12295.168} C_VEL
LIN {X 0,Y 375.514,Z 638.615,A -85,B 0,C 180,E1 12298.511,E2 12298.511} C_VEL
LIN {X 0,Y 378.642,Z 655.606,A -85,B 0,C 180,E1 12300.888,E2 12300.888} C_VEL
LIN {X 0,Y 372.687,Z 683.046,A -85,B 0,C 180,E1 12304.523,E2 12304.523} C_VEL
LIN {X 0,Y 366.953,Z 706.04,A -85,B 0,C 180,E1 12308.914,E2 12308.914} C_VEL
LIN {X 0,Y 362.247,Z 723.637,A -85,B 0,C 180,E1 12313.831,E2 12313.831} C_VEL
LIN {X 0,Y 359.188,Z 735.894,A -85,B 0,C 180,E1 12319.105,E2 12319.105} C_VEL
LIN {X 0,Y 357.582,Z 743.51,A -85,B 0,C 180,E1 12325.161,E2 12325.161} C_VEL
LIN {X 0,Y 357.073,Z 745.311,A -85,B 0,C 180,E1 12330.002,E2 12330.002} C_VEL
LIN {X 0,Y 357.615,Z 743.428,A -85,B 0,C 180,E1 12334.843,E2 12334.843} C_VEL
LIN {X 0,Y 359.256,Z 735.71,A -85,B 0,C 180,E1 12340.897,E2 12340.897} C_VEL
LIN {X 0,Y 362.465,Z 722.859,A -85,B 0,C 180,E1 12346.322,E2 12346.322} C_VEL
LIN {X 0,Y 367.387,Z 704.286,A -85,B 0,C 180,E1 12351.38,E2 12351.38} C_VEL
LIN {X 0,Y 372.86,Z 682.413,A -85,B 0,C 180,E1 12355.468,E2 12355.468} C_VEL
LIN {X 0,Y 378.489,Z 656.314,A -85,B 0,C 180,E1 12358.932,E2 12358.932} C_VEL
LIN {X 0,Y 374.959,Z 636.488,A -85,B 0,C 180,E1 12361.672,E2 12361.672} C_VEL
LIN {X 0,Y 366.033,Z 608.896,A -85,B 0,C 180,E1 12365.251,E2 12365.251} C_VEL
LIN {X 0,Y 353.326,Z 580.66,A -85,B 0,C 180,E1 12368.764,E2 12368.764} C_VEL
LIN {X 0,Y 353.207,Z 580.66,A -85,B 0,C 180,E1 12376.576,E2 12376.576} C_VEL
LIN {X 0,Y 353.309,Z 580.66,A -85,B 0,C 180,E1 12384.242,E2 12384.242} C_VEL
LIN {X 0,Y 353.464,Z 580.66,A -85,B 0,C 180,E1 12391.999,E2 12391.999} C_VEL
LIN {X 0,Y 353.833,Z 580.66,A -85,B 0,C 180,E1 12400.058,E2 12400.058} C_VEL
LIN {X 0,Y 354.14,Z 580.66,A -85,B 0,C 180,E1 12407.705,E2 12407.705} C_VEL
LIN {X 0,Y 354.666,Z 580.66,A -85,B 0,C 180,E1 12415.124,E2 12415.124} C_VEL
LIN {X 0,Y 354.922,Z 580.66,A -85,B 0,C 180,E1 12420.005,E2 12420.005} C_VEL
LIN {X 0,Y 354.521,Z 580.66,A -85,B 0,C 180,E1 12427.34,E2 12427.34} C_VEL
LIN {X 0,Y 354.158,Z 580.66,A -85,B 0,C 180,E1 12434.815,E2 12434.815} C_VEL
LIN {X 0,Y 353.744,Z 580.66,A -85,B 0,C 180,E1 12442.58,E2 12442.58} C_VEL
LIN {X 0,Y 353.496,Z 580.66,A -85,B 0,C 180,E1 12448.009,E2 12448.009} C_VEL
LIN {X 0,Y 353.252,Z 580.66,A -85,B 0,C 180,E1 12455.745,E2 12455.745} C_VEL
LIN {X 0,Y 353.18,Z 580.66,A -85,B 0,C 180,E1 12463.42,E2 12463.42} C_VEL
LIN {X 0,Y 353.316,Z 580.756,A -85,B 0,C 180,E1 12464.995,E2 12464.995} C_VEL
LIN {X 0,Y 355.856,Z 586.462,A -85,B 0,C 180,E1 12465.52,E2 12465.52} C_VEL
LIN {X 0,Y 376.267,Z 626.738,A -85,B 0,C 180,E1 12469.239,E2 12469.239} C_VEL
LIN {X 0,Y 385.292,Z 651.302,A -85,B 0,C 180,E1 12471.139,E2 12471.139} C_VEL
LIN {X 0,Y 380.509,Z 689.694,A -85,B 0,C 180,E1 12472.921,E2 12472.921} C_VEL
LIN {X 0,Y 374.467,Z 726.094,A -85,B 0,C 180,E1 12475.656,E2 12475.656} C_VEL
LIN {X 0,Y 368.59,Z 758.217,A -85,B 0,C 180,E1 12479.146,E2 12479.146} C_VEL
LIN {X 0,Y 363.06,Z 787.572,A -85,B 0,C 180,E1 12483.579,E2 12483.579} C_VEL
LIN {X 0,Y 359.003,Z 812.441,A -85,B 0,C 180,E1 12488.743,E2 12488.743} C_VEL
LIN {X 0,Y 356.838,Z 830.837,A -85,B 0,C 180,E1 12494.044,E2 12494.044} C_VEL
LIN {X 0,Y 356.151,Z 844.015,A -85,B 0,C 180,E1 12499.625,E2 12499.625} C_VEL
LIN {X 0,Y 356.178,Z 850.506,A -85,B 0,C 180,E1 12504.093,E2 12504.093} C_VEL
LIN {X 0,Y 356.215,Z 853.087,A -85,B 0,C 180,E1 12507.57,E2 12507.57} C_VEL
LIN {X 0,Y 356.32,Z 853.107,A -85,B 0,C 180,E1 12512.425,E2 12512.425} C_VEL
LIN {X 0,Y 356.165,Z 848.913,A -85,B 0,C 180,E1 12517.3,E2 12517.3} C_VEL
LIN {X 0,Y 356.298,Z 838.354,A -85,B 0,C 180,E1 12523.071,E2 12523.071} C_VEL
LIN {X 0,Y 356.353,Z 837.297,A -85,B 0,C 180,E1 12523.509,E2 12523.509} C_VEL
LIN {X 0,Y 355.355,Z 833.994,A -85,B 0,C 180,E1 12524.804,E2 12524.804} C_VEL
LIN {X 0,Y 349.764,Z 823.698,A -85,B 0,C 180,E1 12528.263,E2 12528.263} C_VEL
LIN {X 0,Y 349.766,Z 822.633,A -85,B 0,C 180,E1 12528.58,E2 12528.58} C_VEL
LIN {X 0,Y 352.831,Z 801.612,A -85,B 0,C 180,E1 12533.969,E2 12533.969} C_VEL
LIN {X 0,Y 357.944,Z 774.55,A -85,B 0,C 180,E1 12538.996,E2 12538.996} C_VEL
LIN {X 0,Y 364.245,Z 743.162,A -85,B 0,C 180,E1 12543.175,E2 12543.175} C_VEL
LIN {X 0,Y 370.696,Z 709.417,A -85,B 0,C 180,E1 12546.351,E2 12546.351} C_VEL
LIN {X 0,Y 376.237,Z 674.118,A -85,B 0,C 180,E1 12548.576,E2 12548.576} C_VEL
LIN {X 0,Y 378.363,Z 652.023,A -85,B 0,C 180,E1 12549.577,E2 12549.577} C_VEL
LIN {X 0,Y 365.092,Z 618.793,A -85,B 0,C 180,E1 12552.372,E2 12552.372} C_VEL
LIN {X 0,Y 345.383,Z 581.553,A -85,B 0,C 180,E1 12556.194,E2 12556.194} C_VEL
LIN {X 0,Y 345.329,Z 580.66,A -85,B 0,C 180,E1 12556.88,E2 12556.88} C_VEL
LIN {X 0,Y 345.271,Z 580.66,A -85,B 0,C 180,E1 12562.274,E2 12562.274} C_VEL
LIN {X 0,Y 345.439,Z 580.66,A -85,B 0,C 180,E1 12568.383,E2 12568.383} C_VEL
LIN {X 0,Y 345.723,Z 580.66,A -85,B 0,C 180,E1 12576.421,E2 12576.421} C_VEL
LIN {X 0,Y 346.013,Z 580.66,A -85,B 0,C 180,E1 12583.608,E2 12583.608} C_VEL
LIN {X 0,Y 346.333,Z 580.66,A -85,B 0,C 180,E1 12589.959,E2 12589.959} C_VEL
LIN {X 0,Y 347.003,Z 580.66,A -85,B 0,C 180,E1 12597.503,E2 12597.503} C_VEL
LIN {X 0,Y 346.852,Z 580.66,A -85,B 0,C 180,E1 12604.987,E2 12604.987} C_VEL
LIN {X 0,Y 346.353,Z 580.66,A -85,B 0,C 180,E1 12612.576,E2 12612.576} C_VEL
LIN {X 0,Y 345.905,Z 580.66,A -85,B 0,C 180,E1 12620.419,E2 12620.419} C_VEL
LIN {X 0,Y 345.672,Z 580.66,A -85,B 0,C 180,E1 12625.876,E2 12625.876} C_VEL
LIN {X 0,Y 345.38,Z 580.66,A -85,B 0,C 180,E1 12633.896,E2 12633.896} C_VEL
LIN {X 0,Y 345.189,Z 580.66,A -85,B 0,C 180,E1 12640.964,E2 12640.964} C_VEL
LIN {X 0,Y 345.228,Z 580.66,A -85,B 0,C 180,E1 12647.981,E2 12647.981} C_VEL
LIN {X 0,Y 345.359,Z 580.66,A -85,B 0,C 180,E1 12649.973,E2 12649.973} C_VEL
LIN {X 0,Y 349.855,Z 590.677,A -85,B 0,C 180,E1 12651.176,E2 12651.176} C_VEL
LIN {X 0,Y 361.788,Z 617.812,A -85,B 0,C 180,E1 12654.781,E2 12654.781} C_VEL
LIN {X 0,Y 369.308,Z 643.839,A -85,B 0,C 180,E1 12658.353,E2 12658.353} C_VEL
LIN {X 0,Y 371.75,Z 657.712,A -85,B 0,C 180,E1 12660.387,E2 12660.387} C_VEL
LIN {X 0,Y 365.676,Z 684.319,A -85,B 0,C 180,E1 12663.999,E2 12663.999} C_VEL
LIN {X 0,Y 359.665,Z 707.269,A -85,B 0,C 180,E1 12668.466,E2 12668.466} C_VEL
LIN {X 0,Y 354.795,Z 724.618,A -85,B 0,C 180,E1 12673.401,E2 12673.401} C_VEL
LIN {X 0,Y 351.505,Z 737.089,A -85,B 0,C 180,E1 12678.864,E2 12678.864} C_VEL
LIN {X 0,Y 350.01,Z 743.642,A -85,B 0,C 180,E1 12683.815,E2 12683.815} C_VEL
LIN {X 0,Y 349.618,Z 745.98,A -85,B 0,C 180,E1 12687.528,E2 12687.528} C_VEL
LIN {X 0,Y 349.629,Z 745.938,A -85,B 0,C 180,E1 12692.476,E2 12692.476} C_VEL
LIN {X 0,Y 350.575,Z 741.386,A -85,B 0,C 180,E1 12698.179,E2 12698.179} C_VEL
LIN {X 0,Y 352.841,Z 731.948,A -85,B 0,C 180,E1 12703.606,E2 12703.606} C_VEL
LIN {X 0,Y 357.19,Z 716.258,A -85,B 0,C 180,E1 12709.113,E2 12709.113} C_VEL
LIN {X 0,Y 362.774,Z 695.587,A -85,B 0,C 180,E1 12713.912,E2 12713.912} C_VEL
LIN {X 0,Y 368.986,Z 670.046,A -85,B 0,C 180,E1 12717.996,E2 12717.996} C_VEL
LIN {X 0,Y 371.75,Z 655.838,A -85,B 0,C 180,E1 12719.749,E2 12719.749} C_VEL
LIN {X 0,Y 365.498,Z 629.098,A -85,B 0,C 180,E1 12723.58,E2 12723.58} C_VEL
LIN {X 0,Y 355.061,Z 601.227,A -85,B 0,C 180,E1 12727.293,E2 12727.293} C_VEL
LIN {X 0,Y 345.32,Z 580.66,A -85,B 0,C 180,E1 12730.033,E2 12730.033} C_VEL
LIN {X 0,Y 345.214,Z 580.66,A -85,B 0,C 180,E1 12737.996,E2 12737.996} C_VEL
LIN {X 0,Y 345.346,Z 580.66,A -85,B 0,C 180,E1 12745.396,E2 12745.396} C_VEL
LIN {X 0,Y 345.452,Z 580.66,A -85,B 0,C 180,E1 12751.29,E2 12751.29} C_VEL
LIN {X 0,Y 345.733,Z 580.66,A -85,B 0,C 180,E1 12756.877,E2 12756.877} C_VEL
LIN {X 0,Y 346.056,Z 580.66,A -85,B 0,C 180,E1 12764.839,E2 12764.839} C_VEL
LIN {X 0,Y 346.564,Z 580.66,A -85,B 0,C 180,E1 12772.5,E2 12772.5} C_VEL
LIN {X 0,Y 347.027,Z 580.66,A -85,B 0,C 180,E1 12777.513,E2 12777.513} C_VEL
LIN {X 0,Y 346.754,Z 580.66,A -85,B 0,C 180,E1 12784.997,E2 12784.997} C_VEL
LIN {X 0,Y 346.377,Z 580.66,A -85,B 0,C 180,E1 12792.585,E2 12792.585} C_VEL
LIN {X 0,Y 345.891,Z 580.66,A -85,B 0,C 180,E1 12800.43,E2 12800.43} C_VEL
LIN {X 0,Y 345.663,Z 580.66,A -85,B 0,C 180,E1 12805.887,E2 12805.887} C_VEL
LIN {X 0,Y 345.37,Z 580.66,A -85,B 0,C 180,E1 12813.886,E2 12813.886} C_VEL
LIN {X 0,Y 345.18,Z 580.66,A -85,B 0,C 180,E1 12821.998,E2 12821.998} C_VEL
LIN {X 0,Y 345.317,Z 581.226,A -85,B 0,C 180,E1 12823.812,E2 12823.812} C_VEL
LIN {X 0,Y 368.68,Z 626.396,A -85,B 0,C 180,E1 12828.322,E2 12828.322} C_VEL
LIN {X 0,Y 378.661,Z 653.203,A -85,B 0,C 180,E1 12830.523,E2 12830.523} C_VEL
LIN {X 0,Y 373.485,Z 691.507,A -85,B 0,C 180,E1 12832.396,E2 12832.396} C_VEL
LIN {X 0,Y 367.487,Z 726.118,A -85,B 0,C 180,E1 12835.083,E2 12835.083} C_VEL
LIN {X 0,Y 361,Z 759.701,A -85,B 0,C 180,E1 12838.865,E2 12838.865} C_VEL
LIN {X 0,Y 355.263,Z 788.531,A -85,B 0,C 180,E1 12843.41,E2 12843.41} C_VEL
LIN {X 0,Y 351.192,Z 812.434,A -85,B 0,C 180,E1 12848.577,E2 12848.577} C_VEL
LIN {X 0,Y 348.896,Z 831.292,A -85,B 0,C 180,E1 12854.316,E2 12854.316} C_VEL
LIN {X 0,Y 348.289,Z 843.884,A -85,B 0,C 180,E1 12860.018,E2 12860.018} C_VEL
LIN {X 0,Y 348.399,Z 850.314,A -85,B 0,C 180,E1 12865.029,E2 12865.029} C_VEL
LIN {X 0,Y 348.485,Z 852.493,A -85,B 0,C 180,E1 12869.998,E2 12869.998} C_VEL
LIN {X 0,Y 348.404,Z 850.278,A -85,B 0,C 180,E1 12875.024,E2 12875.024} C_VEL
LIN {X 0,Y 348.303,Z 842.802,A -85,B 0,C 180,E1 12880.608,E2 12880.608} C_VEL
LIN {X 0,Y 349.026,Z 829.597,A -85,B 0,C 180,E1 12886.318,E2 12886.318} C_VEL
LIN {X 0,Y 349.766,Z 822.633,A -85,B 0,C 180,E1 12888.58,E2 12888.58} C_VEL
LIN {X 0,Y 347.014,Z 814.1,A -85,B 0,C 180,E1 12891.053,E2 12891.053} C_VEL
LIN {X 0,Y 344.545,Z 804.806,A -85,B 0,C 180,E1 12893.501,E2 12893.501} C_VEL
LIN {X 0,Y 349.556,Z 778.882,A -85,B 0,C 180,E1 12898.698,E2 12898.698} C_VEL
LIN {X 0,Y 356.04,Z 748.544,A -85,B 0,C 180,E1 12903.096,E2 12903.096} C_VEL
LIN {X 0,Y 362.49,Z 716.675,A -85,B 0,C 180,E1 12906.38,E2 12906.38} C_VEL
LIN {X 0,Y 368.294,Z 682.929,A -85,B 0,C 180,E1 12908.791,E2 12908.791} C_VEL
LIN {X 0,Y 371.646,Z 653.767,A -85,B 0,C 180,E1 12910.241,E2 12910.241} C_VEL
LIN {X 0,Y 358.4,Z 620.734,A -85,B 0,C 180,E1 12913.191,E2 12913.191} C_VEL
LIN {X 0,Y 339.392,Z 585.894,A -85,B 0,C 180,E1 12917.012,E2 12917.012} C_VEL
LIN {X 0,Y 337.375,Z 580.66,A -85,B 0,C 180,E1 12917.591,E2 12917.591} C_VEL
LIN {X 0,Y 337.352,Z 580.66,A -85,B 0,C 180,E1 12924.442,E2 12924.442} C_VEL
LIN {X 0,Y 337.536,Z 580.66,A -85,B 0,C 180,E1 12930.541,E2 12930.541} C_VEL
LIN {X 0,Y 337.818,Z 580.66,A -85,B 0,C 180,E1 12936.292,E2 12936.292} C_VEL
LIN {X 0,Y 338.016,Z 580.66,A -85,B 0,C 180,E1 12941.787,E2 12941.787} C_VEL
LIN {X 0,Y 338.394,Z 580.66,A -85,B 0,C 180,E1 12949.721,E2 12949.721} C_VEL
LIN {X 0,Y 339.084,Z 580.66,A -85,B 0,C 180,E1 12957.445,E2 12957.445} C_VEL
LIN {X 0,Y 338.921,Z 580.66,A -85,B 0,C 180,E1 12965.104,E2 12965.104} C_VEL
LIN {X 0,Y 338.426,Z 580.66,A -85,B 0,C 180,E1 12972.876,E2 12972.876} C_VEL
LIN {X 0,Y 337.921,Z 580.66,A -85,B 0,C 180,E1 12980.924,E2 12980.924} C_VEL
LIN {X 0,Y 337.645,Z 580.66,A -85,B 0,C 180,E1 12986.652,E2 12986.652} C_VEL
LIN {X 0,Y 337.448,Z 580.66,A -85,B 0,C 180,E1 12992.444,E2 12992.444} C_VEL
LIN {X 0,Y 337.261,Z 580.66,A -85,B 0,C 180,E1 13000.488,E2 13000.488} C_VEL
LIN {X 0,Y 337.335,Z 580.66,A -85,B 0,C 180,E1 13007.862,E2 13007.862} C_VEL
LIN {X 0,Y 337.349,Z 580.66,A -85,B 0,C 180,E1 13008.672,E2 13008.672} C_VEL
LIN {X 0,Y 339.601,Z 586.124,A -85,B 0,C 180,E1 13009.318,E2 13009.318} C_VEL
LIN {X 0,Y 352.114,Z 612.362,A -85,B 0,C 180,E1 13012.994,E2 13012.994} C_VEL
LIN {X 0,Y 360.853,Z 638.901,A -85,B 0,C 180,E1 13016.741,E2 13016.741} C_VEL
LIN {X 0,Y 364.739,Z 660.236,A -85,B 0,C 180,E1 13019.919,E2 13019.919} C_VEL
LIN {X 0,Y 358.697,Z 685.591,A -85,B 0,C 180,E1 13023.454,E2 13023.454} C_VEL
LIN {X 0,Y 352.403,Z 708.497,A -85,B 0,C 180,E1 13027.999,E2 13027.999} C_VEL
LIN {X 0,Y 347.16,Z 726.33,A -85,B 0,C 180,E1 13033.207,E2 13033.207} C_VEL
LIN {X 0,Y 343.834,Z 738.283,A -85,B 0,C 180,E1 13038.612,E2 13038.612} C_VEL
LIN {X 0,Y 342.043,Z 745.88,A -85,B 0,C 180,E1 13044.94,E2 13044.94} C_VEL
LIN {X 0,Y 341.454,Z 747.684,A -85,B 0,C 180,E1 13050.002,E2 13050.002} C_VEL
LIN {X 0,Y 342.076,Z 745.801,A -85,B 0,C 180,E1 13055.063,E2 13055.063} C_VEL
LIN {X 0,Y 343.646,Z 739.135,A -85,B 0,C 180,E1 13060.757,E2 13060.757} C_VEL
LIN {X 0,Y 346.902,Z 727.495,A -85,B 0,C 180,E1 13066.253,E2 13066.253} C_VEL
LIN {X 0,Y 351.789,Z 710.549,A -85,B 0,C 180,E1 13071.384,E2 13071.384} C_VEL
LIN {X 0,Y 357.934,Z 688.604,A -85,B 0,C 180,E1 13075.939,E2 13075.939} C_VEL
LIN {X 0,Y 363.924,Z 663.526,A -85,B 0,C 180,E1 13079.582,E2 13079.582} C_VEL
LIN {X 0,Y 364.378,Z 656.201,A -85,B 0,C 180,E1 13080.568,E2 13080.568} C_VEL
LIN {X 0,Y 358.251,Z 629.745,A -85,B 0,C 180,E1 13084.462,E2 13084.462} C_VEL
LIN {X 0,Y 347.313,Z 601.2,A -85,B 0,C 180,E1 13088.439,E2 13088.439} C_VEL
LIN {X 0,Y 337.34,Z 581.433,A -85,B 0,C 180,E1 13091.169,E2 13091.169} C_VEL
LIN {X 0,Y 337.324,Z 580.66,A -85,B 0,C 180,E1 13097.866,E2 13097.866} C_VEL
LIN {X 0,Y 337.311,Z 580.66,A -85,B 0,C 180,E1 13104.449,E2 13104.449} C_VEL
LIN {X 0,Y 337.507,Z 580.66,A -85,B 0,C 180,E1 13110.549,E2 13110.549} C_VEL
LIN {X 0,Y 337.799,Z 580.66,A -85,B 0,C 180,E1 13116.302,E2 13116.302} C_VEL
LIN {X 0,Y 337.993,Z 580.66,A -85,B 0,C 180,E1 13121.796,E2 13121.796} C_VEL
LIN {X 0,Y 338.382,Z 580.66,A -85,B 0,C 180,E1 13129.731,E2 13129.731} C_VEL
LIN {X 0,Y 339.108,Z 580.66,A -85,B 0,C 180,E1 13137.455,E2 13137.455} C_VEL
LIN {X 0,Y 338.829,Z 580.66,A -85,B 0,C 180,E1 13145.115,E2 13145.115} C_VEL
LIN {X 0,Y 338.449,Z 580.66,A -85,B 0,C 180,E1 13152.885,E2 13152.885} C_VEL
LIN {X 0,Y 337.915,Z 580.66,A -85,B 0,C 180,E1 13160.934,E2 13160.934} C_VEL
LIN {X 0,Y 337.631,Z 580.66,A -85,B 0,C 180,E1 13166.637,E2 13166.637} C_VEL
LIN {X 0,Y 337.453,Z 580.66,A -85,B 0,C 180,E1 13172.455,E2 13172.455} C_VEL
LIN {X 0,Y 337.244,Z 580.66,A -85,B 0,C 180,E1 13180.478,E2 13180.478} C_VEL
LIN {X 0,Y 337.352,Z 581.269,A -85,B 0,C 180,E1 13182.539,E2 13182.539} C_VEL
LIN {X 0,Y 360.341,Z 624.724,A -85,B 0,C 180,E1 13187.212,E2 13187.212} C_VEL
LIN {X 0,Y 371.939,Z 654.99,A -85,B 0,C 180,E1 13189.865,E2 13189.865} C_VEL
LIN {X 0,Y 366.722,Z 692.158,A -85,B 0,C 180,E1 13191.778,E2 13191.778} C_VEL
LIN {X 0,Y 360.319,Z 727.177,A -85,B 0,C 180,E1 13194.581,E2 13194.581} C_VEL
LIN {X 0,Y 353.572,Z 760.172,A -85,B 0,C 180,E1 13198.437,E2 13198.437} C_VEL
LIN {X 0,Y 347.56,Z 788.999,A -85,B 0,C 180,E1 13203.142,E2 13203.142} C_VEL
LIN {X 0,Y 343.314,Z 812.616,A -85,B 0,C 180,E1 13208.479,E2 13208.479} C_VEL
LIN {X 0,Y 341.088,Z 830.033,A -85,B 0,C 180,E1 13213.947,E2 13213.947} C_VEL
LIN {X 0,Y 340.445,Z 842.662,A -85,B 0,C 180,E1 13219.786,E2 13219.786} C_VEL
LIN {X 0,Y 340.578,Z 849.119,A -85,B 0,C 180,E1 13224.914,E2 13224.914} C_VEL
LIN {X 0,Y 340.687,Z 851.308,A -85,B 0,C 180,E1 13229.998,E2 13229.998} C_VEL
LIN {X 0,Y 340.575,Z 849.127,A -85,B 0,C 180,E1 13235.081,E2 13235.081} C_VEL
LIN {X 0,Y 340.447,Z 841.578,A -85,B 0,C 180,E1 13240.855,E2 13240.855} C_VEL
LIN {X 0,Y 341.233,Z 828.338,A -85,B 0,C 180,E1 13246.702,E2 13246.702} C_VEL
LIN {X 0,Y 343.852,Z 809.211,A -85,B 0,C 180,E1 13252.41,E2 13252.41} C_VEL
LIN {X 0,Y 344.545,Z 804.806,A -85,B 0,C 180,E1 13253.501,E2 13253.501} C_VEL
LIN {X 0,Y 342.549,Z 794.827,A -85,B 0,C 180,E1 13255.889,E2 13255.889} C_VEL
LIN {X 0,Y 341.034,Z 783.988,A -85,B 0,C 180,E1 13258.192,E2 13258.192} C_VEL
LIN {X 0,Y 347.538,Z 754.592,A -85,B 0,C 180,E1 13262.866,E2 13262.866} C_VEL
LIN {X 0,Y 354.264,Z 723.307,A -85,B 0,C 180,E1 13266.416,E2 13266.416} C_VEL
LIN {X 0,Y 360.903,Z 688.191,A -85,B 0,C 180,E1 13269.175,E2 13269.175} C_VEL
LIN {X 0,Y 365.203,Z 656.529,A -85,B 0,C 180,E1 13270.834,E2 13270.834} C_VEL
LIN {X 0,Y 352.771,Z 624.687,A -85,B 0,C 180,E1 13273.83,E2 13273.83} C_VEL
LIN {X 0,Y 334.539,Z 591.023,A -85,B 0,C 180,E1 13277.654,E2 13277.654} C_VEL
LIN {X 0,Y 329.559,Z 582.278,A -85,B 0,C 180,E1 13278.796,E2 13278.796} C_VEL
LIN {X 0,Y 329.391,Z 580.66,A -85,B 0,C 180,E1 13278.995,E2 13278.995} C_VEL
LIN {X 0,Y 329.44,Z 580.66,A -85,B 0,C 180,E1 13286.654,E2 13286.654} C_VEL
LIN {X 0,Y 329.678,Z 580.66,A -85,B 0,C 180,E1 13292.757,E2 13292.757} C_VEL
LIN {X 0,Y 329.927,Z 580.66,A -85,B 0,C 180,E1 13298.534,E2 13298.534} C_VEL
LIN {X 0,Y 330.337,Z 580.66,A -85,B 0,C 180,E1 13306.793,E2 13306.793} C_VEL
LIN {X 0,Y 330.884,Z 580.66,A -85,B 0,C 180,E1 13314.762,E2 13314.762} C_VEL
LIN {X 0,Y 331.251,Z 580.66,A -85,B 0,C 180,E1 13319.995,E2 13319.995} C_VEL
LIN {X 0,Y 331.018,Z 580.66,A -85,B 0,C 180,E1 13325.226,E2 13325.226} C_VEL
LIN {X 0,Y 330.465,Z 580.66,A -85,B 0,C 180,E1 13333.192,E2 13333.192} C_VEL
LIN {X 0,Y 329.942,Z 580.66,A -85,B 0,C 180,E1 13341.455,E2 13341.455} C_VEL
LIN {X 0,Y 329.625,Z 580.66,A -85,B 0,C 180,E1 13349.574,E2 13349.574} C_VEL
LIN {X 0,Y 329.351,Z 580.66,A -85,B 0,C 180,E1 13356.547,E2 13356.547} C_VEL
LIN {X 0,Y 329.362,Z 580.66,A -85,B 0,C 180,E1 13363.4,E2 13363.4} C_VEL
LIN {X 0,Y 329.428,Z 581.358,A -85,B 0,C 180,E1 13367.328,E2 13367.328} C_VEL
LIN {X 0,Y 344.282,Z 611.658,A -85,B 0,C 180,E1 13371.761,E2 13371.761} C_VEL
LIN {X 0,Y 353.501,Z 639.035,A -85,B 0,C 180,E1 13375.779,E2 13375.779} C_VEL
LIN {X 0,Y 357.917,Z 662.056,A -85,B 0,C 180,E1 13379.355,E2 13379.355} C_VEL
LIN {X 0,Y 351.269,Z 688.678,A -85,B 0,C 180,E1 13383.192,E2 13383.192} C_VEL
LIN {X 0,Y 344.797,Z 710.958,A -85,B 0,C 180,E1 13387.826,E2 13387.826} C_VEL
LIN {X 0,Y 339.378,Z 728.645,A -85,B 0,C 180,E1 13393.241,E2 13393.241} C_VEL
LIN {X 0,Y 335.914,Z 740.508,A -85,B 0,C 180,E1 13398.996,E2 13398.996} C_VEL
LIN {X 0,Y 334.272,Z 747.065,A -85,B 0,C 180,E1 13404.822,E2 13404.822} C_VEL
LIN {X 0,Y 333.645,Z 748.87,A -85,B 0,C 180,E1 13410.002,E2 13410.002} C_VEL
LIN {X 0,Y 334.306,Z 746.987,A -85,B 0,C 180,E1 13415.181,E2 13415.181} C_VEL
LIN {X 0,Y 336.228,Z 739.298,A -85,B 0,C 180,E1 13421.653,E2 13421.653} C_VEL
LIN {X 0,Y 339.896,Z 726.868,A -85,B 0,C 180,E1 13427.3,E2 13427.3} C_VEL
LIN {X 0,Y 345.303,Z 709.302,A -85,B 0,C 180,E1 13432.482,E2 13432.482} C_VEL
LIN {X 0,Y 351.406,Z 688.07,A -85,B 0,C 180,E1 13436.801,E2 13436.801} C_VEL
LIN {X 0,Y 357.924,Z 661.356,A -85,B 0,C 180,E1 13440.639,E2 13440.639} C_VEL
LIN {X 0,Y 352.319,Z 634.912,A -85,B 0,C 180,E1 13444.729,E2 13444.729} C_VEL
LIN {X 0,Y 342.706,Z 608.188,A -85,B 0,C 180,E1 13448.629,E2 13448.629} C_VEL
LIN {X 0,Y 329.44,Z 581.541,A -85,B 0,C 180,E1 13452.536,E2 13452.536} C_VEL
LIN {X 0,Y 329.386,Z 580.66,A -85,B 0,C 180,E1 13452.874,E2 13452.874} C_VEL
LIN {X 0,Y 329.364,Z 580.66,A -85,B 0,C 180,E1 13460.113,E2 13460.113} C_VEL
LIN {X 0,Y 329.405,Z 580.66,A -85,B 0,C 180,E1 13466.662,E2 13466.662} C_VEL
LIN {X 0,Y 329.634,Z 580.66,A -85,B 0,C 180,E1 13472.764,E2 13472.764} C_VEL
LIN {X 0,Y 329.92,Z 580.66,A -85,B 0,C 180,E1 13478.544,E2 13478.544} C_VEL
LIN {X 0,Y 330.295,Z 580.66,A -85,B 0,C 180,E1 13486.802,E2 13486.802} C_VEL
LIN {X 0,Y 330.903,Z 580.66,A -85,B 0,C 180,E1 13494.772,E2 13494.772} C_VEL
LIN {X 0,Y 331.219,Z 580.66,A -85,B 0,C 180,E1 13500.005,E2 13500.005} C_VEL
LIN {X 0,Y 330.721,Z 580.66,A -85,B 0,C 180,E1 13507.872,E2 13507.872} C_VEL
LIN {X 0,Y 330.272,Z 580.66,A -85,B 0,C 180,E1 13515.914,E2 13515.914} C_VEL
LIN {X 0,Y 329.811,Z 580.66,A -85,B 0,C 180,E1 13524.32,E2 13524.32} C_VEL
LIN {X 0,Y 329.581,Z 580.66,A -85,B 0,C 180,E1 13530.244,E2 13530.244} C_VEL
LIN {X 0,Y 329.333,Z 580.66,A -85,B 0,C 180,E1 13538.837,E2 13538.837} C_VEL
LIN {X 0,Y 329.362,Z 580.979,A -85,B 0,C 180,E1 13541.159,E2 13541.159} C_VEL
LIN {X 0,Y 331.942,Z 586.504,A -85,B 0,C 180,E1 13541.788,E2 13541.788} C_VEL
LIN {X 0,Y 350.962,Z 620.77,A -85,B 0,C 180,E1 13545.809,E2 13545.809} C_VEL
LIN {X 0,Y 364.245,Z 653.344,A -85,B 0,C 180,E1 13548.893,E2 13548.893} C_VEL
LIN {X 0,Y 365.108,Z 660.603,A -85,B 0,C 180,E1 13549.404,E2 13549.404} C_VEL
LIN {X 0,Y 359.047,Z 698.173,A -85,B 0,C 180,E1 13551.498,E2 13551.498} C_VEL
LIN {X 0,Y 352.089,Z 733.572,A -85,B 0,C 180,E1 13554.631,E2 13554.631} C_VEL
LIN {X 0,Y 345.131,Z 765.625,A -85,B 0,C 180,E1 13558.721,E2 13558.721} C_VEL
LIN {X 0,Y 339.169,Z 792.885,A -85,B 0,C 180,E1 13563.582,E2 13563.582} C_VEL
LIN {X 0,Y 334.997,Z 815.812,A -85,B 0,C 180,E1 13569.222,E2 13569.222} C_VEL
LIN {X 0,Y 333.018,Z 832.148,A -85,B 0,C 180,E1 13574.896,E2 13574.896} C_VEL
LIN {X 0,Y 332.625,Z 843.488,A -85,B 0,C 180,E1 13580.862,E2 13580.862} C_VEL
LIN {X 0,Y 332.663,Z 849.008,A -85,B 0,C 180,E1 13586.32,E2 13586.32} C_VEL
LIN {X 0,Y 332.872,Z 850.121,A -85,B 0,C 180,E1 13589.998,E2 13589.998} C_VEL
LIN {X 0,Y 332.759,Z 847.934,A -85,B 0,C 180,E1 13595.201,E2 13595.201} C_VEL
LIN {X 0,Y 332.604,Z 840.432,A -85,B 0,C 180,E1 13601.069,E2 13601.069} C_VEL
LIN {X 0,Y 333.437,Z 827.171,A -85,B 0,C 180,E1 13607.069,E2 13607.069} C_VEL
LIN {X 0,Y 336.383,Z 807.297,A -85,B 0,C 180,E1 13613.099,E2 13613.099} C_VEL
LIN {X 0,Y 341.034,Z 783.988,A -85,B 0,C 180,E1 13618.192,E2 13618.192} C_VEL
LIN {X 0,Y 339.837,Z 772.656,A -85,B 0,C 180,E1 13620.439,E2 13620.439} C_VEL
LIN {X 0,Y 338.997,Z 760.527,A -85,B 0,C 180,E1 13622.569,E2 13622.569} C_VEL
LIN {X 0,Y 345.824,Z 730.379,A -85,B 0,C 180,E1 13626.355,E2 13626.355} C_VEL
LIN {X 0,Y 353.192,Z 694.704,A -85,B 0,C 180,E1 13629.454,E2 13629.454} C_VEL
LIN {X 0,Y 358.546,Z 658.512,A -85,B 0,C 180,E1 13631.513,E2 13631.513} C_VEL
LIN {X 0,Y 346.359,Z 627,A -85,B 0,C 180,E1 13634.666,E2 13634.666} C_VEL
LIN {X 0,Y 327.805,Z 592.497,A -85,B 0,C 180,E1 13638.776,E2 13638.776} C_VEL
LIN {X 0,Y 321.512,Z 581.425,A -85,B 0,C 180,E1 13640.31,E2 13640.31} C_VEL
LIN {X 0,Y 321.484,Z 580.66,A -85,B 0,C 180,E1 13647.651,E2 13647.651} C_VEL
LIN {X 0,Y 321.807,Z 580.66,A -85,B 0,C 180,E1 13655.035,E2 13655.035} C_VEL
LIN {X 0,Y 322.086,Z 580.66,A -85,B 0,C 180,E1 13660.852,E2 13660.852} C_VEL
LIN {X 0,Y 322.562,Z 580.66,A -85,B 0,C 180,E1 13669.211,E2 13669.211} C_VEL
LIN {X 0,Y 323.244,Z 580.66,A -85,B 0,C 180,E1 13677.32,E2 13677.32} C_VEL
LIN {X 0,Y 323.209,Z 580.66,A -85,B 0,C 180,E1 13682.671,E2 13682.671} C_VEL
LIN {X 0,Y 322.615,Z 580.66,A -85,B 0,C 180,E1 13690.839,E2 13690.839} C_VEL
LIN {X 0,Y 322.322,Z 580.66,A -85,B 0,C 180,E1 13696.307,E2 13696.307} C_VEL
LIN {X 0,Y 321.998,Z 580.66,A -85,B 0,C 180,E1 13702.011,E2 13702.011} C_VEL
LIN {X 0,Y 321.72,Z 580.66,A -85,B 0,C 180,E1 13707.964,E2 13707.964} C_VEL
LIN {X 0,Y 321.46,Z 580.66,A -85,B 0,C 180,E1 13714.275,E2 13714.275} C_VEL
LIN {X 0,Y 321.339,Z 580.66,A -85,B 0,C 180,E1 13721.299,E2 13721.299} C_VEL
LIN {X 0,Y 321.397,Z 580.66,A -85,B 0,C 180,E1 13725.768,E2 13725.768} C_VEL
LIN {X 0,Y 323.803,Z 586.269,A -85,B 0,C 180,E1 13726.525,E2 13726.525} C_VEL
LIN {X 0,Y 337.085,Z 612.561,A -85,B 0,C 180,E1 13730.696,E2 13730.696} C_VEL
LIN {X 0,Y 346.448,Z 640.115,A -85,B 0,C 180,E1 13734.921,E2 13734.921} C_VEL
LIN {X 0,Y 350.979,Z 663.441,A -85,B 0,C 180,E1 13738.682,E2 13738.682} C_VEL
LIN {X 0,Y 344.338,Z 689.946,A -85,B 0,C 180,E1 13742.608,E2 13742.608} C_VEL
LIN {X 0,Y 337.563,Z 712.183,A -85,B 0,C 180,E1 13747.325,E2 13747.325} C_VEL
LIN {X 0,Y 332.115,Z 729.083,A -85,B 0,C 180,E1 13752.551,E2 13752.551} C_VEL
LIN {X 0,Y 328.23,Z 741.703,A -85,B 0,C 180,E1 13758.735,E2 13758.735} C_VEL
LIN {X 0,Y 326.489,Z 748.252,A -85,B 0,C 180,E1 13764.699,E2 13764.699} C_VEL
LIN {X 0,Y 325.855,Z 750.053,A -85,B 0,C 180,E1 13770.002,E2 13770.002} C_VEL
LIN {X 0,Y 326.524,Z 748.176,A -85,B 0,C 180,E1 13775.305,E2 13775.305} C_VEL
LIN {X 0,Y 328.585,Z 740.491,A -85,B 0,C 180,E1 13781.928,E2 13781.928} C_VEL
LIN {X 0,Y 332.536,Z 727.777,A -85,B 0,C 180,E1 13787.81,E2 13787.81} C_VEL
LIN {X 0,Y 338.114,Z 710.526,A -85,B 0,C 180,E1 13792.987,E2 13792.987} C_VEL
LIN {X 0,Y 344.466,Z 689.347,A -85,B 0,C 180,E1 13797.386,E2 13797.386} C_VEL
LIN {X 0,Y 350.838,Z 662.78,A -85,B 0,C 180,E1 13801.327,E2 13801.327} C_VEL
LIN {X 0,Y 345.752,Z 637.701,A -85,B 0,C 180,E1 13805.352,E2 13805.352} C_VEL
LIN {X 0,Y 336.197,Z 610.658,A -85,B 0,C 180,E1 13809.478,E2 13809.478} C_VEL
LIN {X 0,Y 323.281,Z 585.684,A -85,B 0,C 180,E1 13813.476,E2 13813.476} C_VEL
LIN {X 0,Y 321.39,Z 580.66,A -85,B 0,C 180,E1 13814.143,E2 13814.143} C_VEL
LIN {X 0,Y 321.427,Z 580.66,A -85,B 0,C 180,E1 13822.399,E2 13822.399} C_VEL
LIN {X 0,Y 321.521,Z 580.66,A -85,B 0,C 180,E1 13828.927,E2 13828.927} C_VEL
LIN {X 0,Y 321.781,Z 580.66,A -85,B 0,C 180,E1 13835.044,E2 13835.044} C_VEL
LIN {X 0,Y 322.071,Z 580.66,A -85,B 0,C 180,E1 13840.862,E2 13840.862} C_VEL
LIN {X 0,Y 322.546,Z 580.66,A -85,B 0,C 180,E1 13849.25,E2 13849.25} C_VEL
LIN {X 0,Y 323.267,Z 580.66,A -85,B 0,C 180,E1 13857.33,E2 13857.33} C_VEL
LIN {X 0,Y 323.139,Z 580.66,A -85,B 0,C 180,E1 13862.681,E2 13862.681} C_VEL
LIN {X 0,Y 322.658,Z 580.66,A -85,B 0,C 180,E1 13870.855,E2 13870.855} C_VEL
LIN {X 0,Y 322.315,Z 580.66,A -85,B 0,C 180,E1 13876.318,E2 13876.318} C_VEL
LIN {X 0,Y 321.995,Z 580.66,A -85,B 0,C 180,E1 13882.022,E2 13882.022} C_VEL
LIN {X 0,Y 321.723,Z 580.66,A -85,B 0,C 180,E1 13887.975,E2 13887.975} C_VEL
LIN {X 0,Y 321.442,Z 580.66,A -85,B 0,C 180,E1 13894.289,E2 13894.289} C_VEL
LIN {X 0,Y 321.419,Z 580.66,A -85,B 0,C 180,E1 13899.669,E2 13899.669} C_VEL
LIN {X 0,Y 323.89,Z 586.357,A -85,B 0,C 180,E1 13900.339,E2 13900.339} C_VEL
LIN {X 0,Y 342.573,Z 619.075,A -85,B 0,C 180,E1 13904.525,E2 13904.525} C_VEL
LIN {X 0,Y 356.069,Z 650.832,A -85,B 0,C 180,E1 13907.761,E2 13907.761} C_VEL
LIN {X 0,Y 358.759,Z 660.581,A -85,B 0,C 180,E1 13908.652,E2 13908.652} C_VEL
LIN {X 0,Y 352.351,Z 698.52,A -85,B 0,C 180,E1 13910.825,E2 13910.825} C_VEL
LIN {X 0,Y 345.447,Z 732.105,A -85,B 0,C 180,E1 13913.845,E2 13913.845} C_VEL
LIN {X 0,Y 338.14,Z 764.184,A -85,B 0,C 180,E1 13917.985,E2 13917.985} C_VEL
LIN {X 0,Y 331.794,Z 791.557,A -85,B 0,C 180,E1 13922.947,E2 13922.947} C_VEL
LIN {X 0,Y 327.344,Z 814.523,A -85,B 0,C 180,E1 13928.713,E2 13928.713} C_VEL
LIN {X 0,Y 325.198,Z 830.899,A -85,B 0,C 180,E1 13934.524,E2 13934.524} C_VEL
LIN {X 0,Y 324.791,Z 842.276,A -85,B 0,C 180,E1 13940.64,E2 13940.64} C_VEL
LIN {X 0,Y 324.926,Z 846.727,A -85,B 0,C 180,E1 13944.669,E2 13944.669} C_VEL
LIN {X 0,Y 325.08,Z 848.937,A -85,B 0,C 180,E1 13949.998,E2 13949.998} C_VEL
LIN {X 0,Y 324.92,Z 846.737,A -85,B 0,C 180,E1 13955.327,E2 13955.327} C_VEL
LIN {X 0,Y 324.737,Z 840.234,A -85,B 0,C 180,E1 13960.709,E2 13960.709} C_VEL
LIN {X 0,Y 325.457,Z 827.707,A -85,B 0,C 180,E1 13966.776,E2 13966.776} C_VEL
LIN {X 0,Y 328.303,Z 809.011,A -85,B 0,C 180,E1 13972.874,E2 13972.874} C_VEL
LIN {X 0,Y 333.426,Z 784.209,A -85,B 0,C 180,E1 13978.56,E2 13978.56} C_VEL
LIN {X 0,Y 338.997,Z 760.527,A -85,B 0,C 180,E1 13982.569,E2 13982.569} C_VEL
LIN {X 0,Y 338.326,Z 747.897,A -85,B 0,C 180,E1 13984.636,E2 13984.636} C_VEL
LIN {X 0,Y 337.637,Z 736.367,A -85,B 0,C 180,E1 13986.352,E2 13986.352} C_VEL
LIN {X 0,Y 337.984,Z 734.578,A -85,B 0,C 180,E1 13986.557,E2 13986.557} C_VEL
LIN {X 0,Y 345.391,Z 701.083,A -85,B 0,C 180,E1 13989.709,E2 13989.709} C_VEL
LIN {X 0,Y 351.729,Z 666.253,A -85,B 0,C 180,E1 13991.869,E2 13991.869} C_VEL
LIN {X 0,Y 351.56,Z 659.191,A -85,B 0,C 180,E1 13992.346,E2 13992.346} C_VEL
LIN {X 0,Y 338.857,Z 626.619,A -85,B 0,C 180,E1 13995.808,E2 13995.808} C_VEL
LIN {X 0,Y 321.274,Z 594.894,A -85,B 0,C 180,E1 13999.898,E2 13999.898} C_VEL
LIN {X 0,Y 313.693,Z 582.102,A -85,B 0,C 180,E1 14001.853,E2 14001.853} C_VEL
LIN {X 0,Y 313.559,Z 580.66,A -85,B 0,C 180,E1 14001.935,E2 14001.935} C_VEL
LIN {X 0,Y 313.627,Z 580.66,A -85,B 0,C 180,E1 14009.994,E2 14009.994} C_VEL
LIN {X 0,Y 313.98,Z 580.66,A -85,B 0,C 180,E1 14017.385,E2 14017.385} C_VEL
LIN {X 0,Y 314.347,Z 580.66,A -85,B 0,C 180,E1 14023.738,E2 14023.738} C_VEL
LIN {X 0,Y 314.818,Z 580.66,A -85,B 0,C 180,E1 14031.728,E2 14031.728} C_VEL
LIN {X 0,Y 315.338,Z 580.66,A -85,B 0,C 180,E1 14037.252,E2 14037.252} C_VEL
LIN {X 0,Y 315.314,Z 580.66,A -85,B 0,C 180,E1 14042.738,E2 14042.738} C_VEL
LIN {X 0,Y 314.708,Z 580.66,A -85,B 0,C 180,E1 14051.051,E2 14051.051} C_VEL
LIN {X 0,Y 314.355,Z 580.66,A -85,B 0,C 180,E1 14056.732,E2 14056.732} C_VEL
LIN {X 0,Y 313.892,Z 580.66,A -85,B 0,C 180,E1 14064.033,E2 14064.033} C_VEL
LIN {X 0,Y 313.59,Z 580.66,A -85,B 0,C 180,E1 14071.95,E2 14071.95} C_VEL
LIN {X 0,Y 313.331,Z 580.66,A -85,B 0,C 180,E1 14079.603,E2 14079.603} C_VEL
LIN {X 0,Y 313.398,Z 581.411,A -85,B 0,C 180,E1 14084.199,E2 14084.199} C_VEL
LIN {X 0,Y 328.87,Z 611.115,A -85,B 0,C 180,E1 14089.195,E2 14089.195} C_VEL
LIN {X 0,Y 338.331,Z 637.301,A -85,B 0,C 180,E1 14093.385,E2 14093.385} C_VEL
LIN {X 0,Y 343.734,Z 662.911,A -85,B 0,C 180,E1 14097.623,E2 14097.623} C_VEL
LIN {X 0,Y 343.363,Z 669.787,A -85,B 0,C 180,E1 14098.68,E2 14098.68} C_VEL
LIN {X 0,Y 336.369,Z 694.609,A -85,B 0,C 180,E1 14102.628,E2 14102.628} C_VEL
LIN {X 0,Y 329.587,Z 715.881,A -85,B 0,C 180,E1 14107.456,E2 14107.456} C_VEL
LIN {X 0,Y 323.993,Z 732.234,A -85,B 0,C 180,E1 14112.939,E2 14112.939} C_VEL
LIN {X 0,Y 320.311,Z 743.905,A -85,B 0,C 180,E1 14119.141,E2 14119.141} C_VEL
LIN {X 0,Y 318.721,Z 749.437,A -85,B 0,C 180,E1 14124.569,E2 14124.569} C_VEL
LIN {X 0,Y 318.046,Z 751.24,A -85,B 0,C 180,E1 14130.002,E2 14130.002} C_VEL
LIN {X 0,Y 318.758,Z 749.362,A -85,B 0,C 180,E1 14135.435,E2 14135.435} C_VEL
LIN {X 0,Y 320.938,Z 741.684,A -85,B 0,C 180,E1 14142.217,E2 14142.217} C_VEL
LIN {X 0,Y 325.319,Z 728.373,A -85,B 0,C 180,E1 14148.456,E2 14148.456} C_VEL
LIN {X 0,Y 331.35,Z 710.485,A -85,B 0,C 180,E1 14153.84,E2 14153.84} C_VEL
LIN {X 0,Y 338.123,Z 688.797,A -85,B 0,C 180,E1 14158.307,E2 14158.307} C_VEL
LIN {X 0,Y 343.867,Z 664.679,A -85,B 0,C 180,E1 14161.957,E2 14161.957} C_VEL
LIN {X 0,Y 338.851,Z 639.421,A -85,B 0,C 180,E1 14166.171,E2 14166.171} C_VEL
LIN {X 0,Y 329.928,Z 613.626,A -85,B 0,C 180,E1 14170.289,E2 14170.289} C_VEL
LIN {X 0,Y 315.901,Z 586.377,A -85,B 0,C 180,E1 14174.892,E2 14174.892} C_VEL
LIN {X 0,Y 313.393,Z 580.66,A -85,B 0,C 180,E1 14175.721,E2 14175.721} C_VEL
LIN {X 0,Y 313.376,Z 580.66,A -85,B 0,C 180,E1 14181.256,E2 14181.256} C_VEL
LIN {X 0,Y 313.586,Z 580.66,A -85,B 0,C 180,E1 14188.049,E2 14188.049} C_VEL
LIN {X 0,Y 313.869,Z 580.66,A -85,B 0,C 180,E1 14195.988,E2 14195.988} C_VEL
LIN {X 0,Y 314.301,Z 580.66,A -85,B 0,C 180,E1 14203.784,E2 14203.784} C_VEL
LIN {X 0,Y 314.821,Z 580.66,A -85,B 0,C 180,E1 14211.738,E2 14211.738} C_VEL
LIN {X 0,Y 315.361,Z 580.66,A -85,B 0,C 180,E1 14217.263,E2 14217.263} C_VEL
LIN {X 0,Y 315.223,Z 580.66,A -85,B 0,C 180,E1 14222.749,E2 14222.749} C_VEL
LIN {X 0,Y 314.749,Z 580.66,A -85,B 0,C 180,E1 14231.06,E2 14231.06} C_VEL
LIN {X 0,Y 314.331,Z 580.66,A -85,B 0,C 180,E1 14236.744,E2 14236.744} C_VEL
LIN {X 0,Y 313.889,Z 580.66,A -85,B 0,C 180,E1 14244.02,E2 14244.02} C_VEL
LIN {X 0,Y 313.595,Z 580.66,A -85,B 0,C 180,E1 14251.962,E2 14251.962} C_VEL
LIN {X 0,Y 313.506,Z 580.66,A -85,B 0,C 180,E1 14258.039,E2 14258.039} C_VEL
LIN {X 0,Y 316.171,Z 586.521,A -85,B 0,C 180,E1 14258.85,E2 14258.85} C_VEL
LIN {X 0,Y 334.95,Z 618.981,A -85,B 0,C 180,E1 14263.328,E2 14263.328} C_VEL
LIN {X 0,Y 348.613,Z 650.235,A -85,B 0,C 180,E1 14266.754,E2 14266.754} C_VEL
LIN {X 0,Y 352.257,Z 662.47,A -85,B 0,C 180,E1 14267.961,E2 14267.961} C_VEL
LIN {X 0,Y 345.715,Z 698.873,A -85,B 0,C 180,E1 14270.127,E2 14270.127} C_VEL
LIN {X 0,Y 338.239,Z 733.531,A -85,B 0,C 180,E1 14273.346,E2 14273.346} C_VEL
LIN {X 0,Y 330.91,Z 763.936,A -85,B 0,C 180,E1 14277.411,E2 14277.411} C_VEL
LIN {X 0,Y 324.482,Z 790.237,A -85,B 0,C 180,E1 14282.286,E2 14282.286} C_VEL
LIN {X 0,Y 319.706,Z 813.234,A -85,B 0,C 180,E1 14288.179,E2 14288.179} C_VEL
LIN {X 0,Y 317.395,Z 829.653,A -85,B 0,C 180,E1 14294.133,E2 14294.133} C_VEL
LIN {X 0,Y 316.939,Z 841.061,A -85,B 0,C 180,E1 14300.406,E2 14300.406} C_VEL
LIN {X 0,Y 317.103,Z 845.532,A -85,B 0,C 180,E1 14304.537,E2 14304.537} C_VEL
LIN {X 0,Y 317.265,Z 847.75,A -85,B 0,C 180,E1 14309.998,E2 14309.998} C_VEL
LIN {X 0,Y 317.097,Z 845.542,A -85,B 0,C 180,E1 14315.459,E2 14315.459} C_VEL
LIN {X 0,Y 316.871,Z 839.01,A -85,B 0,C 180,E1 14320.978,E2 14320.978} C_VEL
LIN {X 0,Y 317.788,Z 825.732,A -85,B 0,C 180,E1 14327.493,E2 14327.493} C_VEL
LIN {X 0,Y 321.003,Z 806.126,A -85,B 0,C 180,E1 14333.874,E2 14333.874} C_VEL
LIN {X 0,Y 326.463,Z 781.726,A -85,B 0,C 180,E1 14339.482,E2 14339.482} C_VEL
LIN {X 0,Y 333.863,Z 751.789,A -85,B 0,C 180,E1 14344.396,E2 14344.396} C_VEL
LIN {X 0,Y 337.984,Z 734.578,A -85,B 0,C 180,E1 14346.557,E2 14346.557} C_VEL
LIN {X 0,Y 337.838,Z 720.686,A -85,B 0,C 180,E1 14348.358,E2 14348.358} C_VEL
LIN {X 0,Y 337.782,Z 706.185,A -85,B 0,C 180,E1 14350.05,E2 14350.05} C_VEL
LIN {X 0,Y 344.925,Z 669.564,A -85,B 0,C 180,E1 14352.499,E2 14352.499} C_VEL
LIN {X 0,Y 345.192,Z 661.906,A -85,B 0,C 180,E1 14353.013,E2 14353.013} C_VEL
LIN {X 0,Y 332.779,Z 629.566,A -85,B 0,C 180,E1 14356.64,E2 14356.64} C_VEL
LIN {X 0,Y 315.841,Z 598.424,A -85,B 0,C 180,E1 14360.834,E2 14360.834} C_VEL
LIN {X 0,Y 305.724,Z 581.89,A -85,B 0,C 180,E1 14363.591,E2 14363.591} C_VEL
LIN {X 0,Y 305.618,Z 580.66,A -85,B 0,C 180,E1 14363.662,E2 14363.662} C_VEL
LIN {X 0,Y 305.741,Z 580.66,A -85,B 0,C 180,E1 14370.422,E2 14370.422} C_VEL
LIN {X 0,Y 306.027,Z 580.66,A -85,B 0,C 180,E1 14376.763,E2 14376.763} C_VEL
LIN {X 0,Y 306.501,Z 580.66,A -85,B 0,C 180,E1 14385.745,E2 14385.745} C_VEL
LIN {X 0,Y 306.871,Z 580.66,A -85,B 0,C 180,E1 14391.512,E2 14391.512} C_VEL
LIN {X 0,Y 307.415,Z 580.66,A -85,B 0,C 180,E1 14397.181,E2 14397.181} C_VEL
LIN {X 0,Y 307.398,Z 580.66,A -85,B 0,C 180,E1 14402.808,E2 14402.808} C_VEL
LIN {X 0,Y 306.777,Z 580.66,A -85,B 0,C 180,E1 14411.341,E2 14411.341} C_VEL
LIN {X 0,Y 306.371,Z 580.66,A -85,B 0,C 180,E1 14417.182,E2 14417.182} C_VEL
LIN {X 0,Y 306.034,Z 580.66,A -85,B 0,C 180,E1 14423.225,E2 14423.225} C_VEL
LIN {X 0,Y 305.726,Z 580.66,A -85,B 0,C 180,E1 14429.567,E2 14429.567} C_VEL
LIN {X 0,Y 305.373,Z 580.66,A -85,B 0,C 180,E1 14437.763,E2 14437.763} C_VEL
LIN {X 0,Y 305.441,Z 580.66,A -85,B 0,C 180,E1 14442.383,E2 14442.383} C_VEL
LIN {X 0,Y 307.763,Z 586.243,A -85,B 0,C 180,E1 14443.232,E2 14443.232} C_VEL
LIN {X 0,Y 320.233,Z 608.695,A -85,B 0,C 180,E1 14447.411,E2 14447.411} C_VEL
LIN {X 0,Y 329.93,Z 633.81,A -85,B 0,C 180,E1 14451.641,E2 14451.641} C_VEL
LIN {X 0,Y 335.732,Z 657.86,A -85,B 0,C 180,E1 14455.723,E2 14455.723} C_VEL
LIN {X 0,Y 336.78,Z 670.931,A -85,B 0,C 180,E1 14457.967,E2 14457.967} C_VEL
LIN {X 0,Y 329.472,Z 695.859,A -85,B 0,C 180,E1 14462.005,E2 14462.005} C_VEL
LIN {X 0,Y 322.388,Z 717.103,A -85,B 0,C 180,E1 14466.924,E2 14466.924} C_VEL
LIN {X 0,Y 316.283,Z 734.12,A -85,B 0,C 180,E1 14472.818,E2 14472.818} C_VEL
LIN {X 0,Y 312.632,Z 745.095,A -85,B 0,C 180,E1 14478.871,E2 14478.871} C_VEL
LIN {X 0,Y 310.942,Z 750.624,A -85,B 0,C 180,E1 14484.433,E2 14484.433} C_VEL
LIN {X 0,Y 310.241,Z 752.425,A -85,B 0,C 180,E1 14490.002,E2 14490.002} C_VEL
LIN {X 0,Y 311.007,Z 750.546,A -85,B 0,C 180,E1 14495.571,E2 14495.571} C_VEL
LIN {X 0,Y 313.289,Z 742.879,A -85,B 0,C 180,E1 14502.52,E2 14502.52} C_VEL
LIN {X 0,Y 317.869,Z 729.682,A -85,B 0,C 180,E1 14508.865,E2 14508.865} C_VEL
LIN {X 0,Y 324.215,Z 711.721,A -85,B 0,C 180,E1 14514.399,E2 14514.399} C_VEL
LIN {X 0,Y 331.28,Z 690.07,A -85,B 0,C 180,E1 14518.946,E2 14518.946} C_VEL
LIN {X 0,Y 337.021,Z 667.19,A -85,B 0,C 180,E1 14522.5,E2 14522.5} C_VEL
LIN {X 0,Y 332.511,Z 643.009,A -85,B 0,C 180,E1 14526.699,E2 14526.699} C_VEL
LIN {X 0,Y 324.161,Z 617.852,A -85,B 0,C 180,E1 14530.907,E2 14530.907} C_VEL
LIN {X 0,Y 311.469,Z 592.257,A -85,B 0,C 180,E1 14535.45,E2 14535.45} C_VEL
LIN {X 0,Y 305.612,Z 582.252,A -85,B 0,C 180,E1 14537.334,E2 14537.334} C_VEL
LIN {X 0,Y 305.455,Z 580.66,A -85,B 0,C 180,E1 14537.515,E2 14537.515} C_VEL
LIN {X 0,Y 305.421,Z 580.66,A -85,B 0,C 180,E1 14543.648,E2 14543.648} C_VEL
LIN {X 0,Y 305.713,Z 580.66,A -85,B 0,C 180,E1 14550.432,E2 14550.432} C_VEL
LIN {X 0,Y 306.014,Z 580.66,A -85,B 0,C 180,E1 14556.774,E2 14556.774} C_VEL
LIN {X 0,Y 306.281,Z 580.66,A -85,B 0,C 180,E1 14562.813,E2 14562.813} C_VEL
LIN {X 0,Y 306.872,Z 580.66,A -85,B 0,C 180,E1 14571.523,E2 14571.523} C_VEL
LIN {X 0,Y 307.438,Z 580.66,A -85,B 0,C 180,E1 14577.192,E2 14577.192} C_VEL
LIN {X 0,Y 307.306,Z 580.66,A -85,B 0,C 180,E1 14582.82,E2 14582.82} C_VEL
LIN {X 0,Y 306.814,Z 580.66,A -85,B 0,C 180,E1 14591.35,E2 14591.35} C_VEL
LIN {X 0,Y 306.348,Z 580.66,A -85,B 0,C 180,E1 14597.194,E2 14597.194} C_VEL
LIN {X 0,Y 306.032,Z 580.66,A -85,B 0,C 180,E1 14603.236,E2 14603.236} C_VEL
LIN {X 0,Y 305.735,Z 580.66,A -85,B 0,C 180,E1 14609.578,E2 14609.578} C_VEL
LIN {X 0,Y 305.59,Z 580.66,A -85,B 0,C 180,E1 14616.341,E2 14616.341} C_VEL
LIN {X 0,Y 307.951,Z 586.306,A -85,B 0,C 180,E1 14617.115,E2 14617.115} C_VEL
LIN {X 0,Y 325.862,Z 615.902,A -85,B 0,C 180,E1 14621.681,E2 14621.681} C_VEL
LIN {X 0,Y 340.097,Z 646.836,A -85,B 0,C 180,E1 14625.381,E2 14625.381} C_VEL
LIN {X 0,Y 345.588,Z 665.372,A -85,B 0,C 180,E1 14627.306,E2 14627.306} C_VEL
LIN {X 0,Y 338.937,Z 700.215,A -85,B 0,C 180,E1 14629.479,E2 14629.479} C_VEL
LIN {X 0,Y 331.007,Z 735.088,A -85,B 0,C 180,E1 14632.847,E2 14632.847} C_VEL
LIN {X 0,Y 323.287,Z 765.313,A -85,B 0,C 180,E1 14637.081,E2 14637.081} C_VEL
LIN {X 0,Y 316.451,Z 792.06,A -85,B 0,C 180,E1 14642.293,E2 14642.293} C_VEL
LIN {X 0,Y 311.698,Z 814.165,A -85,B 0,C 180,E1 14648.336,E2 14648.336} C_VEL
LIN {X 0,Y 309.459,Z 829.92,A -85,B 0,C 180,E1 14654.442,E2 14654.442} C_VEL
LIN {X 0,Y 309.071,Z 839.843,A -85,B 0,C 180,E1 14660.159,E2 14660.159} C_VEL
LIN {X 0,Y 309.265,Z 844.334,A -85,B 0,C 180,E1 14664.398,E2 14664.398} C_VEL
LIN {X 0,Y 309.471,Z 846.566,A -85,B 0,C 180,E1 14669.998,E2 14669.998} C_VEL
LIN {X 0,Y 309.256,Z 844.344,A -85,B 0,C 180,E1 14675.598,E2 14675.598} C_VEL
LIN {X 0,Y 309.011,Z 837.786,A -85,B 0,C 180,E1 14681.261,E2 14681.261} C_VEL
LIN {X 0,Y 310.062,Z 824.483,A -85,B 0,C 180,E1 14687.944,E2 14687.944} C_VEL
LIN {X 0,Y 313.283,Z 805.787,A -85,B 0,C 180,E1 14694.224,E2 14694.224} C_VEL
LIN {X 0,Y 318.795,Z 782.439,A -85,B 0,C 180,E1 14699.798,E2 14699.798} C_VEL
LIN {X 0,Y 326.236,Z 753.906,A -85,B 0,C 180,E1 14704.711,E2 14704.711} C_VEL
LIN {X 0,Y 334.271,Z 721.653,A -85,B 0,C 180,E1 14708.621,E2 14708.621} C_VEL
LIN {X 0,Y 337.782,Z 706.185,A -85,B 0,C 180,E1 14710.05,E2 14710.05} C_VEL
LIN {X 0,Y 337.746,Z 691.212,A -85,B 0,C 180,E1 14711.603,E2 14711.603} C_VEL
LIN {X 0,Y 337.685,Z 675.732,A -85,B 0,C 180,E1 14712.973,E2 14712.973} C_VEL
LIN {X 0,Y 338.872,Z 664.984,A -85,B 0,C 180,E1 14713.645,E2 14713.645} C_VEL
LIN {X 0,Y 327.732,Z 634.62,A -85,B 0,C 180,E1 14717.228,E2 14717.228} C_VEL
LIN {X 0,Y 311.876,Z 604.447,A -85,B 0,C 180,E1 14721.425,E2 14721.425} C_VEL
LIN {X 0,Y 300.046,Z 586.361,A -85,B 0,C 180,E1 14724.748,E2 14724.748} C_VEL
LIN {X 0,Y 297.625,Z 581.395,A -85,B 0,C 180,E1 14725.542,E2 14725.542} C_VEL
LIN {X 0,Y 297.874,Z 580.66,A -85,B 0,C 180,E1 14732.872,E2 14732.872} C_VEL
LIN {X 0,Y 298.182,Z 580.66,A -85,B 0,C 180,E1 14739.249,E2 14739.249} C_VEL
LIN {X 0,Y 298.526,Z 580.66,A -85,B 0,C 180,E1 14745.356,E2 14745.356} C_VEL
LIN {X 0,Y 299.165,Z 580.66,A -85,B 0,C 180,E1 14754.205,E2 14754.205} C_VEL
LIN {X 0,Y 299.65,Z 580.66,A -85,B 0,C 180,E1 14759.995,E2 14759.995} C_VEL
LIN {X 0,Y 299.287,Z 580.66,A -85,B 0,C 180,E1 14765.782,E2 14765.782} C_VEL
LIN {X 0,Y 298.629,Z 580.66,A -85,B 0,C 180,E1 14774.628,E2 14774.628} C_VEL
LIN {X 0,Y 298.209,Z 580.66,A -85,B 0,C 180,E1 14780.738,E2 14780.738} C_VEL
LIN {X 0,Y 297.869,Z 580.66,A -85,B 0,C 180,E1 14787.117,E2 14787.117} C_VEL
LIN {X 0,Y 297.464,Z 580.66,A -85,B 0,C 180,E1 14795.75,E2 14795.75} C_VEL
LIN {X 0,Y 297.506,Z 581.325,A -85,B 0,C 180,E1 14800.511,E2 14800.511} C_VEL
LIN {X 0,Y 300.366,Z 586.775,A -85,B 0,C 180,E1 14801.541,E2 14801.541} C_VEL
LIN {X 0,Y 313.377,Z 610.634,A -85,B 0,C 180,E1 14806.231,E2 14806.231} C_VEL
LIN {X 0,Y 322.786,Z 634.171,A -85,B 0,C 180,E1 14810.458,E2 14810.458} C_VEL
LIN {X 0,Y 328.838,Z 659.292,A -85,B 0,C 180,E1 14814.896,E2 14814.896} C_VEL
LIN {X 0,Y 330.103,Z 672.617,A -85,B 0,C 180,E1 14817.301,E2 14817.301} C_VEL
LIN {X 0,Y 322.09,Z 698.76,A -85,B 0,C 180,E1 14821.687,E2 14821.687} C_VEL
LIN {X 0,Y 314.797,Z 719.467,A -85,B 0,C 180,E1 14826.709,E2 14826.709} C_VEL
LIN {X 0,Y 308.806,Z 735.357,A -85,B 0,C 180,E1 14832.405,E2 14832.405} C_VEL
LIN {X 0,Y 304.969,Z 746.284,A -85,B 0,C 180,E1 14838.588,E2 14838.588} C_VEL
LIN {X 0,Y 303.113,Z 751.95,A -85,B 0,C 180,E1 14844.552,E2 14844.552} C_VEL
LIN {X 0,Y 302.432,Z 753.612,A -85,B 0,C 180,E1 14850.002,E2 14850.002} C_VEL
LIN {X 0,Y 303.25,Z 751.731,A -85,B 0,C 180,E1 14855.714,E2 14855.714} C_VEL
LIN {X 0,Y 305.649,Z 744.074,A -85,B 0,C 180,E1 14862.838,E2 14862.838} C_VEL
LIN {X 0,Y 310.218,Z 731.595,A -85,B 0,C 180,E1 14869.059,E2 14869.059} C_VEL
LIN {X 0,Y 316.661,Z 714.204,A -85,B 0,C 180,E1 14874.644,E2 14874.644} C_VEL
LIN {X 0,Y 324.477,Z 691.341,A -85,B 0,C 180,E1 14879.613,E2 14879.613} C_VEL
LIN {X 0,Y 330.296,Z 670.574,A -85,B 0,C 180,E1 14882.904,E2 14882.904} C_VEL
LIN {X 0,Y 325.986,Z 645.699,A -85,B 0,C 180,E1 14887.402,E2 14887.402} C_VEL
LIN {X 0,Y 318.129,Z 621.371,A -85,B 0,C 180,E1 14891.674,E2 14891.674} C_VEL
LIN {X 0,Y 306.246,Z 596.941,A -85,B 0,C 180,E1 14896.273,E2 14896.273} C_VEL
LIN {X 0,Y 299.226,Z 585.588,A -85,B 0,C 180,E1 14898.661,E2 14898.661} C_VEL
LIN {X 0,Y 297.476,Z 580.66,A -85,B 0,C 180,E1 14899.544,E2 14899.544} C_VEL
LIN {X 0,Y 297.543,Z 580.66,A -85,B 0,C 180,E1 14906.102,E2 14906.102} C_VEL
LIN {X 0,Y 297.847,Z 580.66,A -85,B 0,C 180,E1 14912.881,E2 14912.881} C_VEL
LIN {X 0,Y 298.175,Z 580.66,A -85,B 0,C 180,E1 14919.26,E2 14919.26} C_VEL
LIN {X 0,Y 298.492,Z 580.66,A -85,B 0,C 180,E1 14925.365,E2 14925.365} C_VEL
LIN {X 0,Y 299.18,Z 580.66,A -85,B 0,C 180,E1 14934.216,E2 14934.216} C_VEL
LIN {X 0,Y 299.629,Z 580.66,A -85,B 0,C 180,E1 14940.005,E2 14940.005} C_VEL
LIN {X 0,Y 299.008,Z 580.66,A -85,B 0,C 180,E1 14948.713,E2 14948.713} C_VEL
LIN {X 0,Y 298.479,Z 580.66,A -85,B 0,C 180,E1 14956.145,E2 14956.145} C_VEL
LIN {X 0,Y 297.966,Z 580.66,A -85,B 0,C 180,E1 14964.276,E2 14964.276} C_VEL
LIN {X 0,Y 297.697,Z 580.66,A -85,B 0,C 180,E1 14970.491,E2 14970.491} C_VEL
LIN {X 0,Y 297.539,Z 580.776,A -85,B 0,C 180,E1 14974.462,E2 14974.462} C_VEL
LIN {X 0,Y 299.871,Z 586.242,A -85,B 0,C 180,E1 14975.255,E2 14975.255} C_VEL
LIN {X 0,Y 312.984,Z 606.772,A -85,B 0,C 180,E1 14978.924,E2 14978.924} C_VEL
LIN {X 0,Y 328.315,Z 635.772,A -85,B 0,C 180,E1 14982.954,E2 14982.954} C_VEL
LIN {X 0,Y 338.831,Z 664.846,A -85,B 0,C 180,E1 14986.362,E2 14986.362} C_VEL
LIN {X 0,Y 336.241,Z 682.625,A -85,B 0,C 180,E1 14987.441,E2 14987.441} C_VEL
LIN {X 0,Y 328.67,Z 717.197,A -85,B 0,C 180,E1 14990.215,E2 14990.215} C_VEL
LIN {X 0,Y 320.498,Z 748.86,A -85,B 0,C 180,E1 14993.946,E2 14993.946} C_VEL
LIN {X 0,Y 312.594,Z 777.588,A -85,B 0,C 180,E1 14998.738,E2 14998.738} C_VEL
LIN {X 0,Y 306.598,Z 801.205,A -85,B 0,C 180,E1 15004.246,E2 15004.246} C_VEL
LIN {X 0,Y 302.592,Z 820.868,A -85,B 0,C 180,E1 15010.643,E2 15010.643} C_VEL
LIN {X 0,Y 301.218,Z 834.661,A -85,B 0,C 180,E1 15017.212,E2 15017.212} C_VEL
LIN {X 0,Y 301.325,Z 841.893,A -85,B 0,C 180,E1 15022.806,E2 15022.806} C_VEL
LIN {X 0,Y 301.467,Z 844.756,A -85,B 0,C 180,E1 15027.129,E2 15027.129} C_VEL
LIN {X 0,Y 301.679,Z 845.382,A -85,B 0,C 180,E1 15029.998,E2 15029.998} C_VEL
LIN {X 0,Y 301.42,Z 843.147,A -85,B 0,C 180,E1 15035.744,E2 15035.744} C_VEL
LIN {X 0,Y 301.135,Z 836.559,A -85,B 0,C 180,E1 15041.56,E2 15041.56} C_VEL
LIN {X 0,Y 302.331,Z 823.047,A -85,B 0,C 180,E1 15048.498,E2 15048.498} C_VEL
LIN {X 0,Y 306.111,Z 803.11,A -85,B 0,C 180,E1 15055.242,E2 15055.242} C_VEL
LIN {X 0,Y 312.139,Z 779.403,A -85,B 0,C 180,E1 15060.903,E2 15060.903} C_VEL
LIN {X 0,Y 320.148,Z 750.212,A -85,B 0,C 180,E1 15065.885,E2 15065.885} C_VEL
LIN {X 0,Y 328.286,Z 718.997,A -85,B 0,C 180,E1 15069.62,E2 15069.62} C_VEL
LIN {X 0,Y 335.962,Z 684.179,A -85,B 0,C 180,E1 15072.475,E2 15072.475} C_VEL
LIN {X 0,Y 337.685,Z 675.732,A -85,B 0,C 180,E1 15072.973,E2 15072.973} C_VEL
LIN {X 0,Y 336.913,Z 667.344,A -85,B 0,C 180,E1 15073.757,E2 15073.757} C_VEL
LIN {X 0,Y 326.505,Z 649.307,A -85,B 0,C 180,E1 15076.582,E2 15076.582} C_VEL
LIN {X 0,Y 312.809,Z 619.195,A -85,B 0,C 180,E1 15080.67,E2 15080.67} C_VEL
LIN {X 0,Y 296.687,Z 592.934,A -85,B 0,C 180,E1 15085.306,E2 15085.306} C_VEL
LIN {X 0,Y 291.565,Z 585.79,A -85,B 0,C 180,E1 15086.929,E2 15086.929} C_VEL
LIN {X 0,Y 289.658,Z 580.66,A -85,B 0,C 180,E1 15087.838,E2 15087.838} C_VEL
LIN {X 0,Y 290.017,Z 580.66,A -85,B 0,C 180,E1 15095.398,E2 15095.398} C_VEL
LIN {X 0,Y 290.358,Z 580.66,A -85,B 0,C 180,E1 15101.827,E2 15101.827} C_VEL
LIN {X 0,Y 290.885,Z 580.66,A -85,B 0,C 180,E1 15110.247,E2 15110.247} C_VEL
LIN {X 0,Y 291.592,Z 580.66,A -85,B 0,C 180,E1 15117.028,E2 15117.028} C_VEL
LIN {X 0,Y 291.589,Z 580.66,A -85,B 0,C 180,E1 15122.961,E2 15122.961} C_VEL
LIN {X 0,Y 290.861,Z 580.66,A -85,B 0,C 180,E1 15131.97,E2 15131.97} C_VEL
LIN {X 0,Y 290.311,Z 580.66,A -85,B 0,C 180,E1 15140.688,E2 15140.688} C_VEL
LIN {X 0,Y 289.851,Z 580.66,A -85,B 0,C 180,E1 15147.931,E2 15147.931} C_VEL
LIN {X 0,Y 289.539,Z 580.66,A -85,B 0,C 180,E1 15156.887,E2 15156.887} C_VEL
LIN {X 0,Y 289.528,Z 581.148,A -85,B 0,C 180,E1 15158.376,E2 15158.376} C_VEL
LIN {X 0,Y 291.936,Z 586.396,A -85,B 0,C 180,E1 15159.361,E2 15159.361} C_VEL
LIN {X 0,Y 303.813,Z 606.366,A -85,B 0,C 180,E1 15163.797,E2 15163.797} C_VEL
LIN {X 0,Y 314.482,Z 630.917,A -85,B 0,C 180,E1 15168.552,E2 15168.552} C_VEL
LIN {X 0,Y 321.284,Z 656.523,A -85,B 0,C 180,E1 15173.247,E2 15173.247} C_VEL
LIN {X 0,Y 323.524,Z 674.133,A -85,B 0,C 180,E1 15176.59,E2 15176.59} C_VEL
LIN {X 0,Y 315.23,Z 700.012,A -85,B 0,C 180,E1 15181.013,E2 15181.013} C_VEL
LIN {X 0,Y 307.579,Z 720.816,A -85,B 0,C 180,E1 15186.175,E2 15186.175} C_VEL
LIN {X 0,Y 301.228,Z 736.89,A -85,B 0,C 180,E1 15192.105,E2 15192.105} C_VEL
LIN {X 0,Y 297.311,Z 747.473,A -85,B 0,C 180,E1 15198.29,E2 15198.29} C_VEL
LIN {X 0,Y 295.4,Z 752.996,A -85,B 0,C 180,E1 15204.139,E2 15204.139} C_VEL
LIN {X 0,Y 294.653,Z 754.793,A -85,B 0,C 180,E1 15210.002,E2 15210.002} C_VEL
LIN {X 0,Y 295.487,Z 752.917,A -85,B 0,C 180,E1 15215.864,E2 15215.864} C_VEL
LIN {X 0,Y 298.022,Z 745.268,A -85,B 0,C 180,E1 15223.172,E2 15223.172} C_VEL
LIN {X 0,Y 302.972,Z 732.522,A -85,B 0,C 180,E1 15229.649,E2 15229.649} C_VEL
LIN {X 0,Y 310.02,Z 714.291,A -85,B 0,C 180,E1 15235.561,E2 15235.561} C_VEL
LIN {X 0,Y 317.739,Z 692.607,A -85,B 0,C 180,E1 15240.306,E2 15240.306} C_VEL
LIN {X 0,Y 323.506,Z 673.378,A -85,B 0,C 180,E1 15243.435,E2 15243.435} C_VEL
LIN {X 0,Y 319.528,Z 648.613,A -85,B 0,C 180,E1 15248.1,E2 15248.1} C_VEL
LIN {X 0,Y 311.758,Z 623.821,A -85,B 0,C 180,E1 15252.66,E2 15252.66} C_VEL
LIN {X 0,Y 299.902,Z 598.985,A -85,B 0,C 180,E1 15257.593,E2 15257.593} C_VEL
LIN {X 0,Y 291.633,Z 586.045,A -85,B 0,C 180,E1 15260.591,E2 15260.591} C_VEL
LIN {X 0,Y 289.494,Z 580.66,A -85,B 0,C 180,E1 15261.536,E2 15261.536} C_VEL
LIN {X 0,Y 289.678,Z 580.66,A -85,B 0,C 180,E1 15268.616,E2 15268.616} C_VEL
LIN {X 0,Y 289.998,Z 580.66,A -85,B 0,C 180,E1 15275.409,E2 15275.409} C_VEL
LIN {X 0,Y 290.345,Z 580.66,A -85,B 0,C 180,E1 15281.838,E2 15281.838} C_VEL
LIN {X 0,Y 290.881,Z 580.66,A -85,B 0,C 180,E1 15290.282,E2 15290.282} C_VEL
LIN {X 0,Y 291.614,Z 580.66,A -85,B 0,C 180,E1 15297.04,E2 15297.04} C_VEL
LIN {X 0,Y 291.469,Z 580.66,A -85,B 0,C 180,E1 15302.973,E2 15302.973} C_VEL
LIN {X 0,Y 290.893,Z 580.66,A -85,B 0,C 180,E1 15311.98,E2 15311.98} C_VEL
LIN {X 0,Y 290.3,Z 580.66,A -85,B 0,C 180,E1 15320.668,E2 15320.668} C_VEL
LIN {X 0,Y 289.837,Z 580.66,A -85,B 0,C 180,E1 15327.945,E2 15327.945} C_VEL
LIN {X 0,Y 289.629,Z 581.331,A -85,B 0,C 180,E1 15332.402,E2 15332.402} C_VEL
LIN {X 0,Y 292.296,Z 586.6,A -85,B 0,C 180,E1 15333.354,E2 15333.354} C_VEL
LIN {X 0,Y 305.613,Z 607.004,A -85,B 0,C 180,E1 15337.378,E2 15337.378} C_VEL
LIN {X 0,Y 321.109,Z 636.054,A -85,B 0,C 180,E1 15341.737,E2 15341.737} C_VEL
LIN {X 0,Y 331.799,Z 665.255,A -85,B 0,C 180,E1 15345.398,E2 15345.398} C_VEL
LIN {X 0,Y 332.379,Z 670.742,A -85,B 0,C 180,E1 15345.903,E2 15345.903} C_VEL
LIN {X 0,Y 324.577,Z 706.911,A -85,B 0,C 180,E1 15348.466,E2 15348.466} C_VEL
LIN {X 0,Y 315.925,Z 740.315,A -85,B 0,C 180,E1 15352.083,E2 15352.083} C_VEL
LIN {X 0,Y 307.382,Z 770.378,A -85,B 0,C 180,E1 15356.814,E2 15356.814} C_VEL
LIN {X 0,Y 300.289,Z 795.981,A -85,B 0,C 180,E1 15362.494,E2 15362.494} C_VEL
LIN {X 0,Y 295.422,Z 816.873,A -85,B 0,C 180,E1 15369.048,E2 15369.048} C_VEL
LIN {X 0,Y 293.454,Z 831.685,A -85,B 0,C 180,E1 15375.858,E2 15375.858} C_VEL
LIN {X 0,Y 293.47,Z 840.687,A -85,B 0,C 180,E1 15382.612,E2 15382.612} C_VEL
LIN {X 0,Y 293.634,Z 843.564,A -85,B 0,C 180,E1 15387.052,E2 15387.052} C_VEL
LIN {X 0,Y 293.862,Z 844.195,A -85,B 0,C 180,E1 15389.998,E2 15389.998} C_VEL
LIN {X 0,Y 293.575,Z 841.948,A -85,B 0,C 180,E1 15395.898,E2 15395.898} C_VEL
LIN {X 0,Y 293.275,Z 834.934,A -85,B 0,C 180,E1 15402.144,E2 15402.144} C_VEL
LIN {X 0,Y 294.583,Z 821.79,A -85,B 0,C 180,E1 15409.003,E2 15409.003} C_VEL
LIN {X 0,Y 298.638,Z 802.105,A -85,B 0,C 180,E1 15415.833,E2 15415.833} C_VEL
LIN {X 0,Y 305.073,Z 778.078,A -85,B 0,C 180,E1 15421.7,E2 15421.7} C_VEL
LIN {X 0,Y 313.783,Z 748.004,A -85,B 0,C 180,E1 15426.877,E2 15426.877} C_VEL
LIN {X 0,Y 322.461,Z 715.935,A -85,B 0,C 180,E1 15430.704,E2 15430.704} C_VEL
LIN {X 0,Y 330.383,Z 681.227,A -85,B 0,C 180,E1 15433.497,E2 15433.497} C_VEL
LIN {X 0,Y 332.544,Z 667.746,A -85,B 0,C 180,E1 15434.328,E2 15434.328} C_VEL
LIN {X 0,Y 326.505,Z 649.307,A -85,B 0,C 180,E1 15436.582,E2 15436.582} C_VEL
LIN {X 0,Y 321.164,Z 640.667,A -85,B 0,C 180,E1 15438.042,E2 15438.042} C_VEL
LIN {X 0,Y 310.167,Z 628.403,A -85,B 0,C 180,E1 15440.754,E2 15440.754} C_VEL
LIN {X 0,Y 293.933,Z 600.033,A -85,B 0,C 180,E1 15445.708,E2 15445.708} C_VEL
LIN {X 0,Y 284.355,Z 586.498,A -85,B 0,C 180,E1 15448.937,E2 15448.937} C_VEL
LIN {X 0,Y 281.809,Z 581.603,A -85,B 0,C 180,E1 15449.939,E2 15449.939} C_VEL
LIN {X 0,Y 281.766,Z 580.66,A -85,B 0,C 180,E1 15450.132,E2 15450.132} C_VEL
LIN {X 0,Y 282.183,Z 580.66,A -85,B 0,C 180,E1 15458.013,E2 15458.013} C_VEL
LIN {X 0,Y 282.587,Z 580.66,A -85,B 0,C 180,E1 15464.51,E2 15464.51} C_VEL
LIN {X 0,Y 283.052,Z 580.66,A -85,B 0,C 180,E1 15470.792,E2 15470.792} C_VEL
LIN {X 0,Y 283.663,Z 580.66,A -85,B 0,C 180,E1 15476.945,E2 15476.945} C_VEL
LIN {X 0,Y 283.666,Z 580.66,A -85,B 0,C 180,E1 15483.043,E2 15483.043} C_VEL
LIN {X 0,Y 283.109,Z 580.66,A -85,B 0,C 180,E1 15489.195,E2 15489.195} C_VEL
LIN {X 0,Y 282.606,Z 580.66,A -85,B 0,C 180,E1 15496.049,E2 15496.049} C_VEL
LIN {X 0,Y 282.121,Z 580.66,A -85,B 0,C 180,E1 15504.606,E2 15504.606} C_VEL
LIN {X 0,Y 281.694,Z 580.66,A -85,B 0,C 180,E1 15512.38,E2 15512.38} C_VEL
LIN {X 0,Y 281.617,Z 580.699,A -85,B 0,C 180,E1 15516.011,E2 15516.011} C_VEL
LIN {X 0,Y 283.699,Z 585.98,A -85,B 0,C 180,E1 15516.975,E2 15516.975} C_VEL
LIN {X 0,Y 286.297,Z 589.758,A -85,B 0,C 180,E1 15518,E2 15518} C_VEL
LIN {X 0,Y 297.811,Z 609.344,A -85,B 0,C 180,E1 15522.652,E2 15522.652} C_VEL
LIN {X 0,Y 308.344,Z 634.187,A -85,B 0,C 180,E1 15527.732,E2 15527.732} C_VEL
LIN {X 0,Y 314.806,Z 659.526,A -85,B 0,C 180,E1 15532.606,E2 15532.606} C_VEL
LIN {X 0,Y 316.458,Z 677.386,A -85,B 0,C 180,E1 15536.109,E2 15536.109} C_VEL
LIN {X 0,Y 307.889,Z 702.904,A -85,B 0,C 180,E1 15540.657,E2 15540.657} C_VEL
LIN {X 0,Y 299.595,Z 724.134,A -85,B 0,C 180,E1 15546.242,E2 15546.242} C_VEL
LIN {X 0,Y 292.897,Z 740.41,A -85,B 0,C 180,E1 15552.796,E2 15552.796} C_VEL
LIN {X 0,Y 288.942,Z 750.409,A -85,B 0,C 180,E1 15559.471,E2 15559.471} C_VEL
LIN {X 0,Y 287.3,Z 755.457,A -85,B 0,C 180,E1 15566.992,E2 15566.992} C_VEL
LIN {X 0,Y 287.419,Z 755.043,A -85,B 0,C 180,E1 15574.178,E2 15574.178} C_VEL
LIN {X 0,Y 289.053,Z 750.257,A -85,B 0,C 180,E1 15580.53,E2 15580.53} C_VEL
LIN {X 0,Y 292.952,Z 740.147,A -85,B 0,C 180,E1 15587.23,E2 15587.23} C_VEL
LIN {X 0,Y 299.682,Z 723.781,A -85,B 0,C 180,E1 15593.756,E2 15593.756} C_VEL
LIN {X 0,Y 307.931,Z 702.409,A -85,B 0,C 180,E1 15599.344,E2 15599.344} C_VEL
LIN {X 0,Y 316.643,Z 676.416,A -85,B 0,C 180,E1 15603.93,E2 15603.93} C_VEL
LIN {X 0,Y 313.522,Z 653.451,A -85,B 0,C 180,E1 15608.447,E2 15608.447} C_VEL
LIN {X 0,Y 306.746,Z 629.897,A -85,B 0,C 180,E1 15612.98,E2 15612.98} C_VEL
LIN {X 0,Y 295.714,Z 605.143,A -85,B 0,C 180,E1 15618.087,E2 15618.087} C_VEL
LIN {X 0,Y 284.31,Z 586.563,A -85,B 0,C 180,E1 15622.641,E2 15622.641} C_VEL
LIN {X 0,Y 281.689,Z 581.614,A -85,B 0,C 180,E1 15623.754,E2 15623.754} C_VEL
LIN {X 0,Y 281.635,Z 580.66,A -85,B 0,C 180,E1 15623.898,E2 15623.898} C_VEL
LIN {X 0,Y 281.782,Z 580.66,A -85,B 0,C 180,E1 15631.195,E2 15631.195} C_VEL
LIN {X 0,Y 282.174,Z 580.66,A -85,B 0,C 180,E1 15638.025,E2 15638.025} C_VEL
LIN {X 0,Y 282.559,Z 580.66,A -85,B 0,C 180,E1 15644.52,E2 15644.52} C_VEL
LIN {X 0,Y 283.206,Z 580.66,A -85,B 0,C 180,E1 15653.359,E2 15653.359} C_VEL
LIN {X 0,Y 283.821,Z 580.66,A -85,B 0,C 180,E1 15660.006,E2 15660.006} C_VEL
LIN {X 0,Y 283.126,Z 580.66,A -85,B 0,C 180,E1 15669.206,E2 15669.206} C_VEL
LIN {X 0,Y 282.591,Z 580.66,A -85,B 0,C 180,E1 15676.02,E2 15676.02} C_VEL
LIN {X 0,Y 282.13,Z 580.66,A -85,B 0,C 180,E1 15684.597,E2 15684.597} C_VEL
LIN {X 0,Y 281.727,Z 580.678,A -85,B 0,C 180,E1 15690.057,E2 15690.057} C_VEL
LIN {X 0,Y 283.785,Z 585.962,A -85,B 0,C 180,E1 15690.935,E2 15690.935} C_VEL
LIN {X 0,Y 286.548,Z 589.63,A -85,B 0,C 180,E1 15691.906,E2 15691.906} C_VEL
LIN {X 0,Y 301.03,Z 611.734,A -85,B 0,C 180,E1 15696.535,E2 15696.535} C_VEL
LIN {X 0,Y 315.676,Z 640.358,A -85,B 0,C 180,E1 15701.03,E2 15701.03} C_VEL
LIN {X 0,Y 326.015,Z 669.868,A -85,B 0,C 180,E1 15704.901,E2 15704.901} C_VEL
LIN {X 0,Y 318.472,Z 705.573,A -85,B 0,C 180,E1 15707.51,E2 15707.51} C_VEL
LIN {X 0,Y 309.428,Z 739.165,A -85,B 0,C 180,E1 15711.186,E2 15711.186} C_VEL
LIN {X 0,Y 300.529,Z 769.042,A -85,B 0,C 180,E1 15715.956,E2 15715.956} C_VEL
LIN {X 0,Y 293.18,Z 793.834,A -85,B 0,C 180,E1 15721.525,E2 15721.525} C_VEL
LIN {X 0,Y 288.225,Z 813.689,A -85,B 0,C 180,E1 15727.736,E2 15727.736} C_VEL
LIN {X 0,Y 285.732,Z 829.139,A -85,B 0,C 180,E1 15734.687,E2 15734.687} C_VEL
LIN {X 0,Y 285.536,Z 838.006,A -85,B 0,C 180,E1 15740.876,E2 15740.876} C_VEL
LIN {X 0,Y 285.807,Z 842.373,A -85,B 0,C 180,E1 15746.971,E2 15746.971} C_VEL
LIN {X 0,Y 286.054,Z 843.009,A -85,B 0,C 180,E1 15749.997,E2 15749.997} C_VEL
LIN {X 0,Y 285.714,Z 840.747,A -85,B 0,C 180,E1 15756.061,E2 15756.061} C_VEL
LIN {X 0,Y 285.418,Z 834.108,A -85,B 0,C 180,E1 15762.206,E2 15762.206} C_VEL
LIN {X 0,Y 286.722,Z 821.452,A -85,B 0,C 180,E1 15769.12,E2 15769.12} C_VEL
LIN {X 0,Y 290.917,Z 802.127,A -85,B 0,C 180,E1 15776.157,E2 15776.157} C_VEL
LIN {X 0,Y 297.574,Z 778.47,A -85,B 0,C 180,E1 15782.167,E2 15782.167} C_VEL
LIN {X 0,Y 306.19,Z 750.25,A -85,B 0,C 180,E1 15787.266,E2 15787.266} C_VEL
LIN {X 0,Y 315.493,Z 717.635,A -85,B 0,C 180,E1 15791.344,E2 15791.344} C_VEL
LIN {X 0,Y 323.8,Z 683.214,A -85,B 0,C 180,E1 15794.234,E2 15794.234} C_VEL
LIN {X 0,Y 326.061,Z 670.025,A -85,B 0,C 180,E1 15795.107,E2 15795.107} C_VEL
LIN {X 0,Y 315.556,Z 640.029,A -85,B 0,C 180,E1 15799.047,E2 15799.047} C_VEL
LIN {X 0,Y 310.167,Z 628.403,A -85,B 0,C 180,E1 15800.754,E2 15800.754} C_VEL
LIN {X 0,Y 301.555,Z 619.283,A -85,B 0,C 180,E1 15803.052,E2 15803.052} C_VEL
LIN {X 0,Y 292.936,Z 610.637,A -85,B 0,C 180,E1 15805.514,E2 15805.514} C_VEL
LIN {X 0,Y 280.337,Z 592.051,A -85,B 0,C 180,E1 15809.898,E2 15809.898} C_VEL
LIN {X 0,Y 276.728,Z 586.669,A -85,B 0,C 180,E1 15811.331,E2 15811.331} C_VEL
LIN {X 0,Y 273.954,Z 581.616,A -85,B 0,C 180,E1 15812.549,E2 15812.549} C_VEL
LIN {X 0,Y 273.906,Z 580.66,A -85,B 0,C 180,E1 15812.9,E2 15812.9} C_VEL
LIN {X 0,Y 274.389,Z 580.66,A -85,B 0,C 180,E1 15820.729,E2 15820.729} C_VEL
LIN {X 0,Y 274.84,Z 580.66,A -85,B 0,C 180,E1 15827.309,E2 15827.309} C_VEL
LIN {X 0,Y 275.356,Z 580.66,A -85,B 0,C 180,E1 15833.702,E2 15833.702} C_VEL
LIN {X 0,Y 275.938,Z 580.66,A -85,B 0,C 180,E1 15839.994,E2 15839.994} C_VEL
LIN {X 0,Y 275.458,Z 580.66,A -85,B 0,C 180,E1 15846.284,E2 15846.284} C_VEL
LIN {X 0,Y 274.934,Z 580.66,A -85,B 0,C 180,E1 15852.675,E2 15852.675} C_VEL
LIN {X 0,Y 274.279,Z 580.66,A -85,B 0,C 180,E1 15860.741,E2 15860.741} C_VEL
LIN {X 0,Y 273.844,Z 580.66,A -85,B 0,C 180,E1 15869.722,E2 15869.722} C_VEL
LIN {X 0,Y 273.74,Z 580.66,A -85,B 0,C 180,E1 15873.354,E2 15873.354} C_VEL
LIN {X 0,Y 275.619,Z 585.765,A -85,B 0,C 180,E1 15874.339,E2 15874.339} C_VEL
LIN {X 0,Y 278.365,Z 589.19,A -85,B 0,C 180,E1 15875.519,E2 15875.519} C_VEL
LIN {X 0,Y 290.682,Z 610.153,A -85,B 0,C 180,E1 15880.938,E2 15880.938} C_VEL
LIN {X 0,Y 301.126,Z 633.943,A -85,B 0,C 180,E1 15886.193,E2 15886.193} C_VEL
LIN {X 0,Y 307.69,Z 659.094,A -85,B 0,C 180,E1 15891.254,E2 15891.254} C_VEL
LIN {X 0,Y 309.828,Z 679.378,A -85,B 0,C 180,E1 15895.417,E2 15895.417} C_VEL
LIN {X 0,Y 301.113,Z 704.145,A -85,B 0,C 180,E1 15899.929,E2 15899.929} C_VEL
LIN {X 0,Y 292.465,Z 725.345,A -85,B 0,C 180,E1 15905.625,E2 15905.625} C_VEL
LIN {X 0,Y 285.828,Z 740.666,A -85,B 0,C 180,E1 15911.824,E2 15911.824} C_VEL
LIN {X 0,Y 281.253,Z 751.6,A -85,B 0,C 180,E1 15919.18,E2 15919.18} C_VEL
LIN {X 0,Y 279.494,Z 756.644,A -85,B 0,C 180,E1 15926.908,E2 15926.908} C_VEL
LIN {X 0,Y 279.546,Z 756.6,A -85,B 0,C 180,E1 15933.097,E2 15933.097} C_VEL
LIN {X 0,Y 280.85,Z 752.935,A -85,B 0,C 180,E1 15939.278,E2 15939.278} C_VEL
LIN {X 0,Y 284.307,Z 744.161,A -85,B 0,C 180,E1 15946.148,E2 15946.148} C_VEL
LIN {X 0,Y 290.723,Z 729.247,A -85,B 0,C 180,E1 15952.912,E2 15952.912} C_VEL
LIN {X 0,Y 298.83,Z 709.735,A -85,B 0,C 180,E1 15958.668,E2 15958.668} C_VEL
LIN {X 0,Y 307.807,Z 685.159,A -85,B 0,C 180,E1 15963.567,E2 15963.567} C_VEL
LIN {X 0,Y 309.833,Z 676.702,A -85,B 0,C 180,E1 15965.009,E2 15965.009} C_VEL
LIN {X 0,Y 306.215,Z 652.139,A -85,B 0,C 180,E1 15970.028,E2 15970.028} C_VEL
LIN {X 0,Y 298.7,Z 627.761,A -85,B 0,C 180,E1 15975,E2 15975} C_VEL
LIN {X 0,Y 287.839,Z 604.847,A -85,B 0,C 180,E1 15980.177,E2 15980.177} C_VEL
LIN {X 0,Y 276.788,Z 586.947,A -85,B 0,C 180,E1 15985,E2 15985} C_VEL
LIN {X 0,Y 273.822,Z 582.167,A -85,B 0,C 180,E1 15986.339,E2 15986.339} C_VEL
LIN {X 0,Y 273.683,Z 580.66,A -85,B 0,C 180,E1 15986.55,E2 15986.55} C_VEL
LIN {X 0,Y 273.956,Z 580.66,A -85,B 0,C 180,E1 15993.864,E2 15993.864} C_VEL
LIN {X 0,Y 274.38,Z 580.66,A -85,B 0,C 180,E1 16000.741,E2 16000.741} C_VEL
LIN {X 0,Y 274.794,Z 580.66,A -85,B 0,C 180,E1 16007.318,E2 16007.318} C_VEL
LIN {X 0,Y 275.367,Z 580.66,A -85,B 0,C 180,E1 16013.714,E2 16013.714} C_VEL
LIN {X 0,Y 275.914,Z 580.66,A -85,B 0,C 180,E1 16020.006,E2 16020.006} C_VEL
LIN {X 0,Y 275.2,Z 580.66,A -85,B 0,C 180,E1 16029.473,E2 16029.473} C_VEL
LIN {X 0,Y 274.702,Z 580.66,A -85,B 0,C 180,E1 16035.946,E2 16035.946} C_VEL
LIN {X 0,Y 274.25,Z 580.66,A -85,B 0,C 180,E1 16042.658,E2 16042.658} C_VEL
LIN {X 0,Y 273.87,Z 580.66,A -85,B 0,C 180,E1 16047.444,E2 16047.444} C_VEL
LIN {X 0,Y 275.923,Z 585.971,A -85,B 0,C 180,E1 16048.435,E2 16048.435} C_VEL
LIN {X 0,Y 278.903,Z 589.705,A -85,B 0,C 180,E1 16049.602,E2 16049.602} C_VEL
LIN {X 0,Y 294.087,Z 612.632,A -85,B 0,C 180,E1 16054.925,E2 16054.925} C_VEL
LIN {X 0,Y 308.805,Z 641.085,A -85,B 0,C 180,E1 16059.782,E2 16059.782} C_VEL
LIN {X 0,Y 318.887,Z 669.503,A -85,B 0,C 180,E1 16063.766,E2 16063.766} C_VEL
LIN {X 0,Y 319.386,Z 675.35,A -85,B 0,C 180,E1 16064.389,E2 16064.389} C_VEL
LIN {X 0,Y 310.72,Z 711.166,A -85,B 0,C 180,E1 16067.164,E2 16067.164} C_VEL
LIN {X 0,Y 301.164,Z 744.128,A -85,B 0,C 180,E1 16071.112,E2 16071.112} C_VEL
LIN {X 0,Y 291.839,Z 773.634,A -85,B 0,C 180,E1 16076.23,E2 16076.23} C_VEL
LIN {X 0,Y 284.386,Z 798.158,A -85,B 0,C 180,E1 16082.335,E2 16082.335} C_VEL
LIN {X 0,Y 279.402,Z 818.213,A -85,B 0,C 180,E1 16089.447,E2 16089.447} C_VEL
LIN {X 0,Y 277.626,Z 831.744,A -85,B 0,C 180,E1 16096.642,E2 16096.642} C_VEL
LIN {X 0,Y 277.772,Z 838.276,A -85,B 0,C 180,E1 16102.192,E2 16102.192} C_VEL
LIN {X 0,Y 277.971,Z 841.18,A -85,B 0,C 180,E1 16106.886,E2 16106.886} C_VEL
LIN {X 0,Y 278.235,Z 841.821,A -85,B 0,C 180,E1 16109.997,E2 16109.997} C_VEL
LIN {X 0,Y 277.867,Z 839.548,A -85,B 0,C 180,E1 16116.232,E2 16116.232} C_VEL
LIN {X 0,Y 277.569,Z 832.883,A -85,B 0,C 180,E1 16122.556,E2 16122.556} C_VEL
LIN {X 0,Y 279.052,Z 820.025,A -85,B 0,C 180,E1 16129.75,E2 16129.75} C_VEL
LIN {X 0,Y 283.608,Z 800.849,A -85,B 0,C 180,E1 16136.884,E2 16136.884} C_VEL
LIN {X 0,Y 290.719,Z 777.169,A -85,B 0,C 180,E1 16143.02,E2 16143.02} C_VEL
LIN {X 0,Y 300.104,Z 747.837,A -85,B 0,C 180,E1 16148.368,E2 16148.368} C_VEL
LIN {X 0,Y 309.461,Z 716.177,A -85,B 0,C 180,E1 16152.334,E2 16152.334} C_VEL
LIN {X 0,Y 317.998,Z 682.044,A -85,B 0,C 180,E1 16155.211,E2 16155.211} C_VEL
LIN {X 0,Y 319.633,Z 672.391,A -85,B 0,C 180,E1 16155.877,E2 16155.877} C_VEL
LIN {X 0,Y 309.341,Z 642.282,A -85,B 0,C 180,E1 16160.073,E2 16160.073} C_VEL
LIN {X 0,Y 295.392,Z 614.745,A -85,B 0,C 180,E1 16164.706,E2 16164.706} C_VEL
LIN {X 0,Y 292.936,Z 610.637,A -85,B 0,C 180,E1 16165.514,E2 16165.514} C_VEL
LIN {X 0,Y 286.443,Z 605.081,A -85,B 0,C 180,E1 16167.509,E2 16167.509} C_VEL
LIN {X 0,Y 277.683,Z 599.213,A -85,B 0,C 180,E1 16170.396,E2 16170.396} C_VEL
LIN {X 0,Y 276.053,Z 596.683,A -85,B 0,C 180,E1 16171.053,E2 16171.053} C_VEL
LIN {X 0,Y 269.376,Z 587.085,A -85,B 0,C 180,E1 16173.935,E2 16173.935} C_VEL
LIN {X 0,Y 266.229,Z 582.122,A -85,B 0,C 180,E1 16175.467,E2 16175.467} C_VEL
LIN {X 0,Y 266.097,Z 580.66,A -85,B 0,C 180,E1 16175.62,E2 16175.62} C_VEL
LIN {X 0,Y 266.735,Z 580.66,A -85,B 0,C 180,E1 16184.078,E2 16184.078} C_VEL
LIN {X 0,Y 267.418,Z 580.66,A -85,B 0,C 180,E1 16193.514,E2 16193.514} C_VEL
LIN {X 0,Y 268.032,Z 580.66,A -85,B 0,C 180,E1 16199.994,E2 16199.994} C_VEL
LIN {X 0,Y 267.515,Z 580.66,A -85,B 0,C 180,E1 16206.471,E2 16206.471} C_VEL
LIN {X 0,Y 266.816,Z 580.66,A -85,B 0,C 180,E1 16215.982,E2 16215.982} C_VEL
LIN {X 0,Y 266.052,Z 580.66,A -85,B 0,C 180,E1 16224.852,E2 16224.852} C_VEL
LIN {X 0,Y 265.942,Z 581.331,A -85,B 0,C 180,E1 16230.397,E2 16230.397} C_VEL
LIN {X 0,Y 268.289,Z 586.329,A -85,B 0,C 180,E1 16231.674,E2 16231.674} C_VEL
LIN {X 0,Y 270.834,Z 589.496,A -85,B 0,C 180,E1 16232.913,E2 16232.913} C_VEL
LIN {X 0,Y 282.061,Z 607.974,A -85,B 0,C 180,E1 16238.323,E2 16238.323} C_VEL
LIN {X 0,Y 292.632,Z 630.562,A -85,B 0,C 180,E1 16243.793,E2 16243.793} C_VEL
LIN {X 0,Y 299.595,Z 653.589,A -85,B 0,C 180,E1 16248.739,E2 16248.739} C_VEL
LIN {X 0,Y 302.957,Z 676.354,A -85,B 0,C 180,E1 16253.574,E2 16253.574} C_VEL
LIN {X 0,Y 302.545,Z 683.414,A -85,B 0,C 180,E1 16255.005,E2 16255.005} C_VEL
LIN {X 0,Y 293.132,Z 708.408,A -85,B 0,C 180,E1 16259.878,E2 16259.878} C_VEL
LIN {X 0,Y 284.378,Z 728.749,A -85,B 0,C 180,E1 16265.722,E2 16265.722} C_VEL
LIN {X 0,Y 277.491,Z 743.89,A -85,B 0,C 180,E1 16272.441,E2 16272.441} C_VEL
LIN {X 0,Y 273.591,Z 752.788,A -85,B 0,C 180,E1 16278.873,E2 16278.873} C_VEL
LIN {X 0,Y 271.701,Z 757.83,A -85,B 0,C 180,E1 16286.819,E2 16286.819} C_VEL
LIN {X 0,Y 271.765,Z 757.783,A -85,B 0,C 180,E1 16293.186,E2 16293.186} C_VEL
LIN {X 0,Y 273.155,Z 754.121,A -85,B 0,C 180,E1 16299.542,E2 16299.542} C_VEL
LIN {X 0,Y 277.129,Z 744.638,A -85,B 0,C 180,E1 16307.028,E2 16307.028} C_VEL
LIN {X 0,Y 284.042,Z 729.439,A -85,B 0,C 180,E1 16313.898,E2 16313.898} C_VEL
LIN {X 0,Y 292.579,Z 709.47,A -85,B 0,C 180,E1 16319.764,E2 16319.764} C_VEL
LIN {X 0,Y 301.9,Z 684.987,A -85,B 0,C 180,E1 16324.627,E2 16324.627} C_VEL
LIN {X 0,Y 302.948,Z 677.167,A -85,B 0,C 180,E1 16326.131,E2 16326.131} C_VEL
LIN {X 0,Y 299.7,Z 654.397,A -85,B 0,C 180,E1 16330.967,E2 16330.967} C_VEL
LIN {X 0,Y 292.77,Z 631.202,A -85,B 0,C 180,E1 16335.94,E2 16335.94} C_VEL
LIN {X 0,Y 283.129,Z 610.076,A -85,B 0,C 180,E1 16340.993,E2 16340.993} C_VEL
LIN {X 0,Y 273.307,Z 593.496,A -85,B 0,C 180,E1 16345.701,E2 16345.701} C_VEL
LIN {X 0,Y 269.165,Z 587.185,A -85,B 0,C 180,E1 16347.727,E2 16347.727} C_VEL
LIN {X 0,Y 266.002,Z 582.462,A -85,B 0,C 180,E1 16349.309,E2 16349.309} C_VEL
LIN {X 0,Y 265.844,Z 580.66,A -85,B 0,C 180,E1 16349.696,E2 16349.696} C_VEL
LIN {X 0,Y 266.184,Z 580.66,A -85,B 0,C 180,E1 16356.629,E2 16356.629} C_VEL
LIN {X 0,Y 266.712,Z 580.66,A -85,B 0,C 180,E1 16364.116,E2 16364.116} C_VEL
LIN {X 0,Y 267.427,Z 580.66,A -85,B 0,C 180,E1 16373.527,E2 16373.527} C_VEL
LIN {X 0,Y 268.006,Z 580.66,A -85,B 0,C 180,E1 16380.006,E2 16380.006} C_VEL
LIN {X 0,Y 267.459,Z 580.66,A -85,B 0,C 180,E1 16386.485,E2 16386.485} C_VEL
LIN {X 0,Y 266.977,Z 580.66,A -85,B 0,C 180,E1 16393.072,E2 16393.072} C_VEL
LIN {X 0,Y 266.445,Z 580.66,A -85,B 0,C 180,E1 16399.87,E2 16399.87} C_VEL
LIN {X 0,Y 266.114,Z 581.387,A -85,B 0,C 180,E1 16404.534,E2 16404.534} C_VEL
LIN {X 0,Y 268.677,Z 586.515,A -85,B 0,C 180,E1 16405.852,E2 16405.852} C_VEL
LIN {X 0,Y 271.094,Z 589.378,A -85,B 0,C 180,E1 16406.919,E2 16406.919} C_VEL
LIN {X 0,Y 284.922,Z 610.096,A -85,B 0,C 180,E1 16412.381,E2 16412.381} C_VEL
LIN {X 0,Y 298.164,Z 633.637,A -85,B 0,C 180,E1 16417.057,E2 16417.057} C_VEL
LIN {X 0,Y 309.724,Z 662.394,A -85,B 0,C 180,E1 16421.609,E2 16421.609} C_VEL
LIN {X 0,Y 313.289,Z 676.092,A -85,B 0,C 180,E1 16423.49,E2 16423.49} C_VEL
LIN {X 0,Y 304.368,Z 711.286,A -85,B 0,C 180,E1 16426.291,E2 16426.291} C_VEL
LIN {X 0,Y 294.604,Z 743.392,A -85,B 0,C 180,E1 16430.205,E2 16430.205} C_VEL
LIN {X 0,Y 284.853,Z 772.909,A -85,B 0,C 180,E1 16435.443,E2 16435.443} C_VEL
LIN {X 0,Y 276.718,Z 798.177,A -85,B 0,C 180,E1 16441.942,E2 16441.942} C_VEL
LIN {X 0,Y 271.781,Z 816.953,A -85,B 0,C 180,E1 16448.843,E2 16448.843} C_VEL
LIN {X 0,Y 269.785,Z 830.514,A -85,B 0,C 180,E1 16456.246,E2 16456.246} C_VEL
LIN {X 0,Y 270.055,Z 838.339,A -85,B 0,C 180,E1 16463.581,E2 16463.581} C_VEL
LIN {X 0,Y 270.419,Z 840.634,A -85,B 0,C 180,E1 16469.997,E2 16469.997} C_VEL
LIN {X 0,Y 270.013,Z 838.347,A -85,B 0,C 180,E1 16476.414,E2 16476.414} C_VEL
LIN {X 0,Y 269.727,Z 831.657,A -85,B 0,C 180,E1 16482.928,E2 16482.928} C_VEL
LIN {X 0,Y 271.418,Z 818.778,A -85,B 0,C 180,E1 16490.329,E2 16490.329} C_VEL
LIN {X 0,Y 276.3,Z 799.565,A -85,B 0,C 180,E1 16497.655,E2 16497.655} C_VEL
LIN {X 0,Y 284.197,Z 774.733,A -85,B 0,C 180,E1 16504.178,E2 16504.178} C_VEL
LIN {X 0,Y 294.125,Z 745.077,A -85,B 0,C 180,E1 16509.568,E2 16509.568} C_VEL
LIN {X 0,Y 303.921,Z 713.124,A -85,B 0,C 180,E1 16513.537,E2 16513.537} C_VEL
LIN {X 0,Y 313.02,Z 677.723,A -85,B 0,C 180,E1 16516.43,E2 16516.43} C_VEL
LIN {X 0,Y 312.224,Z 670.905,A -85,B 0,C 180,E1 16517.221,E2 16517.221} C_VEL
LIN {X 0,Y 302.021,Z 641.841,A -85,B 0,C 180,E1 16521.577,E2 16521.577} C_VEL
LIN {X 0,Y 288.531,Z 615.703,A -85,B 0,C 180,E1 16526.406,E2 16526.406} C_VEL
LIN {X 0,Y 276.053,Z 596.683,A -85,B 0,C 180,E1 16531.053,E2 16531.053} C_VEL
LIN {X 0,Y 270.677,Z 591.249,A -85,B 0,C 180,E1 16533.219,E2 16533.219} C_VEL
LIN {X 0,Y 261.051,Z 586.677,A -85,B 0,C 180,E1 16537.436,E2 16537.436} C_VEL
LIN {X 0,Y 258.423,Z 581.648,A -85,B 0,C 180,E1 16539.022,E2 16539.022} C_VEL
LIN {X 0,Y 258.401,Z 580.66,A -85,B 0,C 180,E1 16539.484,E2 16539.484} C_VEL
LIN {X 0,Y 258.923,Z 580.66,A -85,B 0,C 180,E1 16546.514,E2 16546.514} C_VEL
LIN {X 0,Y 259.469,Z 580.66,A -85,B 0,C 180,E1 16553.315,E2 16553.315} C_VEL
LIN {X 0,Y 260.125,Z 580.66,A -85,B 0,C 180,E1 16559.994,E2 16559.994} C_VEL
LIN {X 0,Y 259.35,Z 580.66,A -85,B 0,C 180,E1 16568.497,E2 16568.497} C_VEL
LIN {X 0,Y 258.723,Z 580.66,A -85,B 0,C 180,E1 16576.947,E2 16576.947} C_VEL
LIN {X 0,Y 258.09,Z 580.66,A -85,B 0,C 180,E1 16586.495,E2 16586.495} C_VEL
LIN {X 0,Y 260.665,Z 586.545,A -85,B 0,C 180,E1 16588.441,E2 16588.441} C_VEL
LIN {X 0,Y 263.16,Z 589.187,A -85,B 0,C 180,E1 16589.787,E2 16589.787} C_VEL
LIN {X 0,Y 274.299,Z 606.936,A -85,B 0,C 180,E1 16595.757,E2 16595.757} C_VEL
LIN {X 0,Y 285.475,Z 630.483,A -85,B 0,C 180,E1 16601.961,E2 16601.961} C_VEL
LIN {X 0,Y 292.623,Z 653.357,A -85,B 0,C 180,E1 16607.212,E2 16607.212} C_VEL
LIN {X 0,Y 296.212,Z 676.389,A -85,B 0,C 180,E1 16612.321,E2 16612.321} C_VEL
LIN {X 0,Y 295.812,Z 685.761,A -85,B 0,C 180,E1 16614.313,E2 16614.313} C_VEL
LIN {X 0,Y 286.409,Z 709.641,A -85,B 0,C 180,E1 16619.094,E2 16619.094} C_VEL
LIN {X 0,Y 277.288,Z 729.95,A -85,B 0,C 180,E1 16625.059,E2 16625.059} C_VEL
LIN {X 0,Y 269.876,Z 745.471,A -85,B 0,C 180,E1 16632.161,E2 16632.161} C_VEL
LIN {X 0,Y 265.915,Z 753.979,A -85,B 0,C 180,E1 16638.547,E2 16638.547} C_VEL
LIN {X 0,Y 263.919,Z 759.014,A -85,B 0,C 180,E1 16646.725,E2 16646.725} C_VEL
LIN {X 0,Y 263.984,Z 758.967,A -85,B 0,C 180,E1 16653.28,E2 16653.28} C_VEL
LIN {X 0,Y 266.022,Z 753.832,A -85,B 0,C 180,E1 16661.454,E2 16661.454} C_VEL
LIN {X 0,Y 270.548,Z 743.979,A -85,B 0,C 180,E1 16668.559,E2 16668.559} C_VEL
LIN {X 0,Y 277.873,Z 728.551,A -85,B 0,C 180,E1 16675.32,E2 16675.32} C_VEL
LIN {X 0,Y 287.089,Z 707.689,A -85,B 0,C 180,E1 16681.27,E2 16681.27} C_VEL
LIN {X 0,Y 296.413,Z 682.393,A -85,B 0,C 180,E1 16686.198,E2 16686.198} C_VEL
LIN {X 0,Y 294.138,Z 661.072,A -85,B 0,C 180,E1 16690.963,E2 16690.963} C_VEL
LIN {X 0,Y 288.39,Z 638.694,A -85,B 0,C 180,E1 16695.972,E2 16695.972} C_VEL
LIN {X 0,Y 279.689,Z 617.449,A -85,B 0,C 180,E1 16701.168,E2 16701.168} C_VEL
LIN {X 0,Y 269.638,Z 599.722,A -85,B 0,C 180,E1 16706.447,E2 16706.447} C_VEL
LIN {X 0,Y 265.097,Z 593.066,A -85,B 0,C 180,E1 16708.846,E2 16708.846} C_VEL
LIN {X 0,Y 261.708,Z 587.312,A -85,B 0,C 180,E1 16710.822,E2 16710.822} C_VEL
LIN {X 0,Y 258.306,Z 582.571,A -85,B 0,C 180,E1 16712.777,E2 16712.777} C_VEL
LIN {X 0,Y 258.067,Z 580.66,A -85,B 0,C 180,E1 16713.237,E2 16713.237} C_VEL
LIN {X 0,Y 258.384,Z 580.66,A -85,B 0,C 180,E1 16719.496,E2 16719.496} C_VEL
LIN {X 0,Y 258.886,Z 580.66,A -85,B 0,C 180,E1 16726.525,E2 16726.525} C_VEL
LIN {X 0,Y 259.476,Z 580.66,A -85,B 0,C 180,E1 16733.496,E2 16733.496} C_VEL
LIN {X 0,Y 260.098,Z 580.66,A -85,B 0,C 180,E1 16740.006,E2 16740.006} C_VEL
LIN {X 0,Y 259.341,Z 580.66,A -85,B 0,C 180,E1 16748.446,E2 16748.446} C_VEL
LIN {X 0,Y 258.702,Z 580.66,A -85,B 0,C 180,E1 16756.962,E2 16756.962} C_VEL
LIN {X 0,Y 258.385,Z 580.66,A -85,B 0,C 180,E1 16760.977,E2 16760.977} C_VEL
LIN {X 0,Y 260.223,Z 585.815,A -85,B 0,C 180,E1 16762.24,E2 16762.24} C_VEL
LIN {X 0,Y 263.572,Z 589.521,A -85,B 0,C 180,E1 16763.959,E2 16763.959} C_VEL
LIN {X 0,Y 273.942,Z 604.73,A -85,B 0,C 180,E1 16768.724,E2 16768.724} C_VEL
LIN {X 0,Y 288.104,Z 627.834,A -85,B 0,C 180,E1 16774.27,E2 16774.27} C_VEL
LIN {X 0,Y 300.606,Z 656.208,A -85,B 0,C 180,E1 16779.33,E2 16779.33} C_VEL
LIN {X 0,Y 306.937,Z 678.371,A -85,B 0,C 180,E1 16782.652,E2 16782.652} C_VEL
LIN {X 0,Y 297.615,Z 712.99,A -85,B 0,C 180,E1 16785.546,E2 16785.546} C_VEL
LIN {X 0,Y 287.503,Z 744.743,A -85,B 0,C 180,E1 16789.577,E2 16789.577} C_VEL
LIN {X 0,Y 277.285,Z 773.88,A -85,B 0,C 180,E1 16794.998,E2 16794.998} C_VEL
LIN {X 0,Y 269.079,Z 798.2,A -85,B 0,C 180,E1 16801.53,E2 16801.53} C_VEL
LIN {X 0,Y 263.767,Z 817.474,A -85,B 0,C 180,E1 16809.048,E2 16809.048} C_VEL
LIN {X 0,Y 261.91,Z 830.404,A -85,B 0,C 180,E1 16816.674,E2 16816.674} C_VEL
LIN {X 0,Y 262.203,Z 837.137,A -85,B 0,C 180,E1 16823.388,E2 16823.388} C_VEL
LIN {X 0,Y 262.599,Z 839.446,A -85,B 0,C 180,E1 16829.997,E2 16829.997} C_VEL
LIN {X 0,Y 262.163,Z 837.146,A -85,B 0,C 180,E1 16836.607,E2 16836.607} C_VEL
LIN {X 0,Y 261.966,Z 829.313,A -85,B 0,C 180,E1 16844.167,E2 16844.167} C_VEL
LIN {X 0,Y 264.199,Z 815.754,A -85,B 0,C 180,E1 16851.789,E2 16851.789} C_VEL
LIN {X 0,Y 269.879,Z 795.664,A -85,B 0,C 180,E1 16859.286,E2 16859.286} C_VEL
LIN {X 0,Y 278.663,Z 770.085,A -85,B 0,C 180,E1 16865.862,E2 16865.862} C_VEL
LIN {X 0,Y 288.69,Z 741.122,A -85,B 0,C 180,E1 16870.993,E2 16870.993} C_VEL
LIN {X 0,Y 299.06,Z 708.481,A -85,B 0,C 180,E1 16874.937,E2 16874.937} C_VEL
LIN {X 0,Y 306.847,Z 677.123,A -85,B 0,C 180,E1 16877.526,E2 16877.526} C_VEL
LIN {X 0,Y 297.3,Z 647.539,A -85,B 0,C 180,E1 16882.13,E2 16882.13} C_VEL
LIN {X 0,Y 284.929,Z 622.036,A -85,B 0,C 180,E1 16887.006,E2 16887.006} C_VEL
LIN {X 0,Y 270.963,Z 600.171,A -85,B 0,C 180,E1 16892.634,E2 16892.634} C_VEL
LIN {X 0,Y 265.463,Z 592.749,A -85,B 0,C 180,E1 16895.155,E2 16895.155} C_VEL
LIN {X 0,Y 262.179,Z 587.471,A -85,B 0,C 180,E1 16896.876,E2 16896.876} C_VEL
LIN {X 0,Y 261.051,Z 586.677,A -85,B 0,C 180,E1 16897.436,E2 16897.436} C_VEL
LIN {X 0,Y 254.838,Z 582.123,A -85,B 0,C 180,E1 16900.865,E2 16900.865} C_VEL
LIN {X 0,Y 250.771,Z 580.66,A -85,B 0,C 180,E1 16904.591,E2 16904.591} C_VEL
LIN {X 0,Y 251.534,Z 580.66,A -85,B 0,C 180,E1 16913.103,E2 16913.103} C_VEL
LIN {X 0,Y 252.221,Z 580.66,A -85,B 0,C 180,E1 16919.994,E2 16919.994} C_VEL
LIN {X 0,Y 251.649,Z 580.66,A -85,B 0,C 180,E1 16926.881,E2 16926.881} C_VEL
LIN {X 0,Y 250.824,Z 580.66,A -85,B 0,C 180,E1 16935.744,E2 16935.744} C_VEL
LIN {X 0,Y 250.339,Z 581.238,A -85,B 0,C 180,E1 16942.356,E2 16942.356} C_VEL
LIN {X 0,Y 252.617,Z 586.243,A -85,B 0,C 180,E1 16944.238,E2 16944.238} C_VEL
LIN {X 0,Y 255.7,Z 589.221,A -85,B 0,C 180,E1 16946.203,E2 16946.203} C_VEL
LIN {X 0,Y 259.683,Z 594.857,A -85,B 0,C 180,E1 16948.756,E2 16948.756} C_VEL
LIN {X 0,Y 270.68,Z 613.996,A -85,B 0,C 180,E1 16955.326,E2 16955.326} C_VEL
LIN {X 0,Y 280.419,Z 635.787,A -85,B 0,C 180,E1 16961.373,E2 16961.373} C_VEL
LIN {X 0,Y 286.571,Z 656.888,A -85,B 0,C 180,E1 16966.44,E2 16966.44} C_VEL
LIN {X 0,Y 289.685,Z 679.636,A -85,B 0,C 180,E1 16971.722,E2 16971.722} C_VEL
LIN {X 0,Y 289.083,Z 688.171,A -85,B 0,C 180,E1 16973.614,E2 16973.614} C_VEL
LIN {X 0,Y 279.065,Z 712.389,A -85,B 0,C 180,E1 16978.642,E2 16978.642} C_VEL
LIN {X 0,Y 269.666,Z 732.172,A -85,B 0,C 180,E1 16984.747,E2 16984.747} C_VEL
LIN {X 0,Y 262.052,Z 747.461,A -85,B 0,C 180,E1 16992.116,E2 16992.116} C_VEL
LIN {X 0,Y 257.645,Z 756.623,A -85,B 0,C 180,E1 16999.884,E2 16999.884} C_VEL
LIN {X 0,Y 256.122,Z 760.199,A -85,B 0,C 180,E1 17006.625,E2 17006.625} C_VEL
LIN {X 0,Y 256.181,Z 760.155,A -85,B 0,C 180,E1 17013.38,E2 17013.38} C_VEL
LIN {X 0,Y 258.351,Z 755.025,A -85,B 0,C 180,E1 17021.798,E2 17021.798} C_VEL
LIN {X 0,Y 263.464,Z 744.542,A -85,B 0,C 180,E1 17029.469,E2 17029.469} C_VEL
LIN {X 0,Y 271.317,Z 728.647,A -85,B 0,C 180,E1 17036.421,E2 17036.421} C_VEL
LIN {X 0,Y 281.162,Z 707.402,A -85,B 0,C 180,E1 17042.46,E2 17042.46} C_VEL
LIN {X 0,Y 289.719,Z 684.593,A -85,B 0,C 180,E1 17046.988,E2 17046.988} C_VEL
LIN {X 0,Y 287.838,Z 663.97,A -85,B 0,C 180,E1 17051.803,E2 17051.803} C_VEL
LIN {X 0,Y 282.388,Z 641.775,A -85,B 0,C 180,E1 17057.017,E2 17057.017} C_VEL
LIN {X 0,Y 273.718,Z 620.164,A -85,B 0,C 180,E1 17062.68,E2 17062.68} C_VEL
LIN {X 0,Y 263.292,Z 601.161,A -85,B 0,C 180,E1 17068.788,E2 17068.788} C_VEL
LIN {X 0,Y 258.003,Z 593.487,A -85,B 0,C 180,E1 17071.966,E2 17071.966} C_VEL
LIN {X 0,Y 254.583,Z 587.714,A -85,B 0,C 180,E1 17074.29,E2 17074.29} C_VEL
LIN {X 0,Y 250.574,Z 582.762,A -85,B 0,C 180,E1 17077.082,E2 17077.082} C_VEL
LIN {X 0,Y 250.303,Z 580.66,A -85,B 0,C 180,E1 17077.874,E2 17077.874} C_VEL
LIN {X 0,Y 250.894,Z 580.66,A -85,B 0,C 180,E1 17086.087,E2 17086.087} C_VEL
LIN {X 0,Y 251.54,Z 580.66,A -85,B 0,C 180,E1 17093.504,E2 17093.504} C_VEL
LIN {X 0,Y 252.195,Z 580.66,A -85,B 0,C 180,E1 17100.006,E2 17100.006} C_VEL
